// TIA Portal V15.1 export
// export: Created 2026-01-09T13:45:09.5933512Z, ExportSetting WithDefaults, WithReadOnly, DisplayName Totally Integrated Automation Portal, DisplayVersion V15.1 Update 8, DisplayName TIA Portal Openness, DisplayVersion V15.1 Update 8, DisplayName STEP 7 Professional, DisplayVersion V15.1 Update 8, DisplayName WinCC Advanced, DisplayVersion V15.1 Update 8
ORGANIZATION_BLOCK "Main_P1"   // OB1, LAD, ProgramCycle
TITLE = "Main Program Sweep (Cycle)"
{ S7_Optimized_Access := 'TRUE' }
VERSION : 0.1
// stored: AutoNumber true, CodeModifiedDate 2026-01-04T14:29:42.3003179Z, CompileDate 2026-01-04T14:29:49.7688293Z, ConstantName OB_Main_P1, CreationDate 2024-10-12T12:36:08.0193576Z, EventClass Program cycle, HandleErrorsWithinBlock false, InterfaceModifiedDate 2008-07-21T16:55:08.419547Z, IsConsistent true, IsIECCheckEnabled false, IsKnowHowProtected false, IsWriteProtected false, ModifiedDate 2026-01-04T14:29:42.3003179Z, ParameterModified 2008-07-21T16:55:08.419547Z, PLCSimAdvancedSupport false, PriorityNumber 1, ProcessImagePartNumber 65535, SetENOAutomatically False, StructureModified 2008-07-21T16:55:08.419547Z
   VAR_INPUT
      Initial_Call : Bool;   // Initial call of this OB
      Remanence : Bool;   // =True, if remanent data are available
   END_VAR
   VAR_TEMP   // added for the SCL form of the ladder/FBD networks
      _w1 : Bool;
      _w2 : Bool;
      _w3 : Bool;
      _w4 : Bool;
      _w5 : Bool;
      _w6 : Bool;
   END_VAR
BEGIN

REGION Network 1: MOVE INPUT
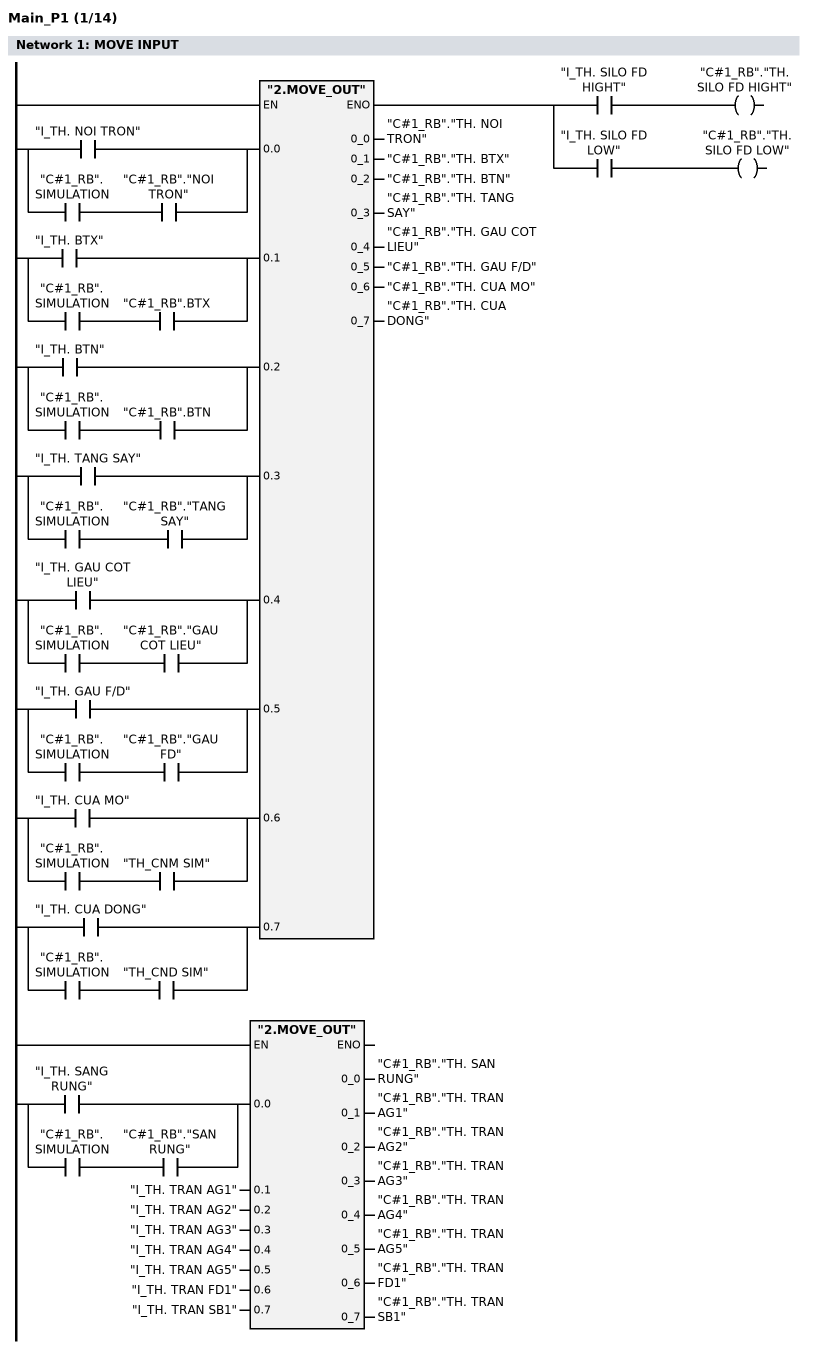
   RUNG wire#powerrail
      "2.MOVE_OUT"("0.0" := wire#w1, "0.1" := wire#w2, "0.2" := wire#w3, "0.3" := wire#w4, "0.4" := wire#w5, "0.5" := wire#w6, "0.6" := wire#w7, "0.7" := wire#w8, "0_0" => "C#1_RB"."TH. NOI TRON", "0_1" => "C#1_RB"."TH. BTX", "0_2" => "C#1_RB"."TH. BTN", "0_3" => "C#1_RB"."TH. TANG SAY", "0_4" => "C#1_RB"."TH. GAU COT LIEU", "0_5" => "C#1_RB"."TH. GAU F/D", "0_6" => "C#1_RB"."TH. CUA MO", "0_7" => "C#1_RB"."TH. CUA DONG")
      wire#w9
      Contact( "I_TH. SILO FD HIGHT" )
      Coil( "C#1_RB"."TH. SILO FD HIGHT" )
   END_RUNG
   RUNG wire#powerrail
      Contact( "I_TH. NOI TRON" )
   END_RUNG wire#w1
   RUNG wire#powerrail
      Contact( "C#1_RB".SIMULATION )
      Contact( "C#1_RB"."NOI TRON" )
   END_RUNG wire#w1
   RUNG wire#powerrail
      Contact( "I_TH. BTX" )
   END_RUNG wire#w2
   RUNG wire#powerrail
      Contact( "C#1_RB".SIMULATION )
      Contact( "C#1_RB".BTX )
   END_RUNG wire#w2
   RUNG wire#powerrail
      Contact( "I_TH. BTN" )
   END_RUNG wire#w3
   RUNG wire#powerrail
      Contact( "C#1_RB".SIMULATION )
      Contact( "C#1_RB".BTN )
   END_RUNG wire#w3
   RUNG wire#powerrail
      Contact( "I_TH. TANG SAY" )
   END_RUNG wire#w4
   RUNG wire#powerrail
      Contact( "C#1_RB".SIMULATION )
      Contact( "C#1_RB"."TANG SAY" )
   END_RUNG wire#w4
   RUNG wire#powerrail
      Contact( "I_TH. GAU COT LIEU" )
   END_RUNG wire#w5
   RUNG wire#powerrail
      Contact( "C#1_RB".SIMULATION )
      Contact( "C#1_RB"."GAU COT LIEU" )
   END_RUNG wire#w5
   RUNG wire#powerrail
      Contact( "I_TH. GAU F/D" )
   END_RUNG wire#w6
   RUNG wire#powerrail
      Contact( "C#1_RB".SIMULATION )
      Contact( "C#1_RB"."GAU FD" )
   END_RUNG wire#w6
   RUNG wire#powerrail
      Contact( "I_TH. CUA MO" )
   END_RUNG wire#w7
   RUNG wire#powerrail
      Contact( "C#1_RB".SIMULATION )
      Contact( "TH_CNM SIM" )
   END_RUNG wire#w7
   RUNG wire#powerrail
      Contact( "I_TH. CUA DONG" )
   END_RUNG wire#w8
   RUNG wire#powerrail
      Contact( "C#1_RB".SIMULATION )
      Contact( "TH_CND SIM" )
   END_RUNG wire#w8
   RUNG wire#w9
      Contact( "I_TH. SILO FD LOW" )
      Coil( "C#1_RB"."TH. SILO FD LOW" )
   END_RUNG
   RUNG wire#powerrail
      "2.MOVE_OUT"("0.0" := wire#w10, "0.1" := "I_TH. TRAN AG1", "0.2" := "I_TH. TRAN AG2", "0.3" := "I_TH. TRAN AG3", "0.4" := "I_TH. TRAN AG4", "0.5" := "I_TH. TRAN AG5", "0.6" := "I_TH. TRAN FD1", "0.7" := "I_TH. TRAN SB1", "0_0" => "C#1_RB"."TH. SAN RUNG", "0_1" => "C#1_RB"."TH. TRAN AG1", "0_2" => "C#1_RB"."TH. TRAN AG2", "0_3" => "C#1_RB"."TH. TRAN AG3", "0_4" => "C#1_RB"."TH. TRAN AG4", "0_5" => "C#1_RB"."TH. TRAN AG5", "0_6" => "C#1_RB"."TH. TRAN FD1", "0_7" => "C#1_RB"."TH. TRAN SB1")
   END_RUNG
   RUNG wire#powerrail
      Contact( "I_TH. SANG RUNG" )
   END_RUNG wire#w10
   RUNG wire#powerrail
      Contact( "C#1_RB".SIMULATION )
      Contact( "C#1_RB"."SAN RUNG" )
   END_RUNG wire#w10
   // the same network as SCL:
   "2.MOVE_OUT"("0.0" := "I_TH. NOI TRON" OR ("C#1_RB".SIMULATION AND "C#1_RB"."NOI TRON"),
                "0.1" := "I_TH. BTX" OR ("C#1_RB".SIMULATION AND "C#1_RB".BTX),
                "0.2" := "I_TH. BTN" OR ("C#1_RB".SIMULATION AND "C#1_RB".BTN),
                "0.3" := "I_TH. TANG SAY" OR ("C#1_RB".SIMULATION AND "C#1_RB"."TANG SAY"),
                "0.4" := "I_TH. GAU COT LIEU" OR ("C#1_RB".SIMULATION AND "C#1_RB"."GAU COT LIEU"),
                "0.5" := "I_TH. GAU F/D" OR ("C#1_RB".SIMULATION AND "C#1_RB"."GAU FD"),
                "0.6" := "I_TH. CUA MO" OR ("C#1_RB".SIMULATION AND "TH_CNM SIM"),
                "0.7" := "I_TH. CUA DONG" OR ("C#1_RB".SIMULATION AND "TH_CND SIM"),
                "0_0" => "C#1_RB"."TH. NOI TRON",
                "0_1" => "C#1_RB"."TH. BTX",
                "0_2" => "C#1_RB"."TH. BTN",
                "0_3" => "C#1_RB"."TH. TANG SAY",
                "0_4" => "C#1_RB"."TH. GAU COT LIEU",
                "0_5" => "C#1_RB"."TH. GAU F/D",
                "0_6" => "C#1_RB"."TH. CUA MO",
                "0_7" => "C#1_RB"."TH. CUA DONG",
                ENO => #_w1);
   "C#1_RB"."TH. SILO FD HIGHT" := #_w1 AND "I_TH. SILO FD HIGHT";
   "C#1_RB"."TH. SILO FD LOW" := #_w1 AND "I_TH. SILO FD LOW";
   "2.MOVE_OUT"("0.0" := "I_TH. SANG RUNG" OR ("C#1_RB".SIMULATION AND "C#1_RB"."SAN RUNG"),
                "0.1" := "I_TH. TRAN AG1",
                "0.2" := "I_TH. TRAN AG2",
                "0.3" := "I_TH. TRAN AG3",
                "0.4" := "I_TH. TRAN AG4",
                "0.5" := "I_TH. TRAN AG5",
                "0.6" := "I_TH. TRAN FD1",
                "0.7" := "I_TH. TRAN SB1",
                "0_0" => "C#1_RB"."TH. SAN RUNG",
                "0_1" => "C#1_RB"."TH. TRAN AG1",
                "0_2" => "C#1_RB"."TH. TRAN AG2",
                "0_3" => "C#1_RB"."TH. TRAN AG3",
                "0_4" => "C#1_RB"."TH. TRAN AG4",
                "0_5" => "C#1_RB"."TH. TRAN AG5",
                "0_6" => "C#1_RB"."TH. TRAN FD1",
                "0_7" => "C#1_RB"."TH. TRAN SB1");
END_REGION

REGION Network 2: MOVE OUTPUT
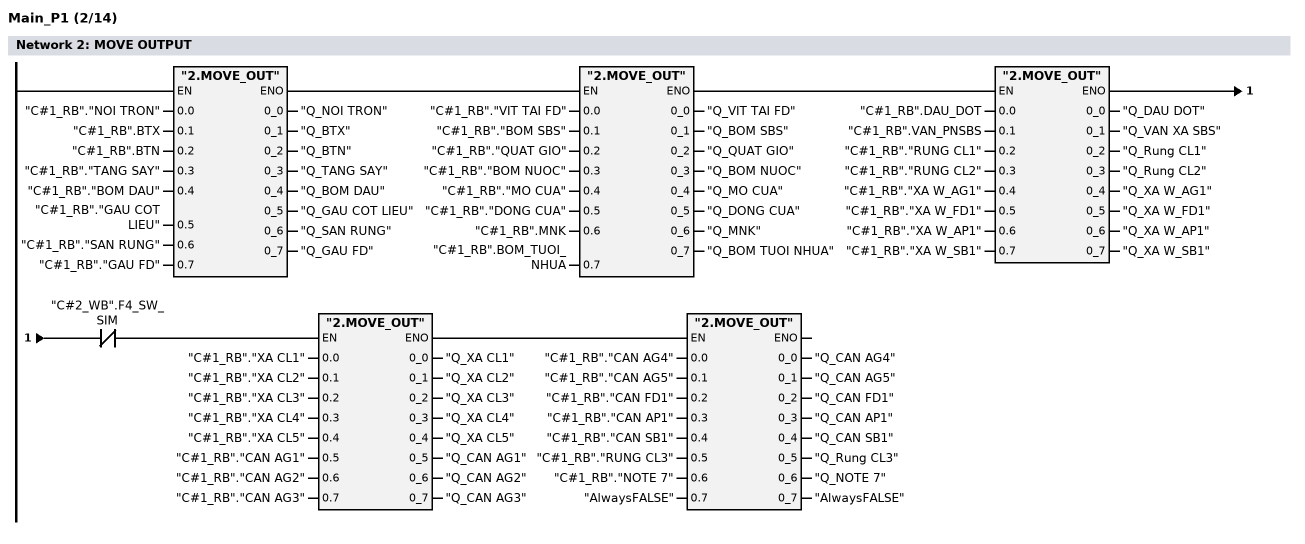
   RUNG wire#powerrail
      "2.MOVE_OUT"("0.0" := "C#1_RB"."NOI TRON", "0.1" := "C#1_RB".BTX, "0.2" := "C#1_RB".BTN, "0.3" := "C#1_RB"."TANG SAY", "0.4" := "C#1_RB"."BOM DAU", "0.5" := "C#1_RB"."GAU COT LIEU", "0.6" := "C#1_RB"."SAN RUNG", "0.7" := "C#1_RB"."GAU FD", "0_0" => "Q_NOI TRON", "0_1" => "Q_BTX", "0_2" => "Q_BTN", "0_3" => "Q_TANG SAY", "0_4" => "Q_BOM DAU", "0_5" => "Q_GAU COT LIEU", "0_6" => "Q_SAN RUNG", "0_7" => "Q_GAU FD")
      "2.MOVE_OUT"("0.0" := "C#1_RB"."VIT TAI FD", "0.1" := "C#1_RB"."BOM SBS", "0.2" := "C#1_RB"."QUAT GIO", "0.3" := "C#1_RB"."BOM NUOC", "0.4" := "C#1_RB"."MO CUA", "0.5" := "C#1_RB"."DONG CUA", "0.6" := "C#1_RB".MNK, "0.7" := "C#1_RB".BOM_TUOI_NHUA, "0_0" => "Q_VIT TAI FD", "0_1" => "Q_BOM SBS", "0_2" => "Q_QUAT GIO", "0_3" => "Q_BOM NUOC", "0_4" => "Q_MO CUA", "0_5" => "Q_DONG CUA", "0_6" => "Q_MNK", "0_7" => "Q_BOM TUOI NHUA")
      "2.MOVE_OUT"("0.0" := "C#1_RB".DAU_DOT, "0.1" := "C#1_RB".VAN_PNSBS, "0.2" := "C#1_RB"."RUNG CL1", "0.3" := "C#1_RB"."RUNG CL2", "0.4" := "C#1_RB"."XA W_AG1", "0.5" := "C#1_RB"."XA W_FD1", "0.6" := "C#1_RB"."XA W_AP1", "0.7" := "C#1_RB"."XA W_SB1", "0_0" => "Q_DAU DOT", "0_1" => "Q_VAN XA SBS", "0_2" => "Q_Rung CL1", "0_3" => "Q_Rung CL2", "0_4" => "Q_XA W_AG1", "0_5" => "Q_XA W_FD1", "0_6" => "Q_XA W_AP1", "0_7" => "Q_XA W_SB1")
      I_Contact( "C#2_WB".F4_SW_SIM )
      "2.MOVE_OUT"("0.0" := "C#1_RB"."XA CL1", "0.1" := "C#1_RB"."XA CL2", "0.2" := "C#1_RB"."XA CL3", "0.3" := "C#1_RB"."XA CL4", "0.4" := "C#1_RB"."XA CL5", "0.5" := "C#1_RB"."CAN AG1", "0.6" := "C#1_RB"."CAN AG2", "0.7" := "C#1_RB"."CAN AG3", "0_0" => "Q_XA CL1", "0_1" => "Q_XA CL2", "0_2" => "Q_XA CL3", "0_3" => "Q_XA CL4", "0_4" => "Q_XA CL5", "0_5" => "Q_CAN AG1", "0_6" => "Q_CAN AG2", "0_7" => "Q_CAN AG3")
      "2.MOVE_OUT"("0.0" := "C#1_RB"."CAN AG4", "0.1" := "C#1_RB"."CAN AG5", "0.2" := "C#1_RB"."CAN FD1", "0.3" := "C#1_RB"."CAN AP1", "0.4" := "C#1_RB"."CAN SB1", "0.5" := "C#1_RB"."RUNG CL3", "0.6" := "C#1_RB"."NOTE 7", "0.7" := "AlwaysFALSE", "0_0" => "Q_CAN AG4", "0_1" => "Q_CAN AG5", "0_2" => "Q_CAN FD1", "0_3" => "Q_CAN AP1", "0_4" => "Q_CAN SB1", "0_5" => "Q_Rung CL3", "0_6" => "Q_NOTE 7", "0_7" => "AlwaysFALSE")
   END_RUNG
   // the same network as SCL:
   "2.MOVE_OUT"("0.0" := "C#1_RB"."NOI TRON",
                "0.1" := "C#1_RB".BTX,
                "0.2" := "C#1_RB".BTN,
                "0.3" := "C#1_RB"."TANG SAY",
                "0.4" := "C#1_RB"."BOM DAU",
                "0.5" := "C#1_RB"."GAU COT LIEU",
                "0.6" := "C#1_RB"."SAN RUNG",
                "0.7" := "C#1_RB"."GAU FD",
                "0_0" => "Q_NOI TRON",
                "0_1" => "Q_BTX",
                "0_2" => "Q_BTN",
                "0_3" => "Q_TANG SAY",
                "0_4" => "Q_BOM DAU",
                "0_5" => "Q_GAU COT LIEU",
                "0_6" => "Q_SAN RUNG",
                "0_7" => "Q_GAU FD",
                ENO => #_w1);
   "2.MOVE_OUT"(EN := #_w1,
                "0.0" := "C#1_RB"."VIT TAI FD",
                "0.1" := "C#1_RB"."BOM SBS",
                "0.2" := "C#1_RB"."QUAT GIO",
                "0.3" := "C#1_RB"."BOM NUOC",
                "0.4" := "C#1_RB"."MO CUA",
                "0.5" := "C#1_RB"."DONG CUA",
                "0.6" := "C#1_RB".MNK,
                "0.7" := "C#1_RB".BOM_TUOI_NHUA,
                "0_0" => "Q_VIT TAI FD",
                "0_1" => "Q_BOM SBS",
                "0_2" => "Q_QUAT GIO",
                "0_3" => "Q_BOM NUOC",
                "0_4" => "Q_MO CUA",
                "0_5" => "Q_DONG CUA",
                "0_6" => "Q_MNK",
                "0_7" => "Q_BOM TUOI NHUA",
                ENO => #_w2);
   "2.MOVE_OUT"(EN := #_w2,
                "0.0" := "C#1_RB".DAU_DOT,
                "0.1" := "C#1_RB".VAN_PNSBS,
                "0.2" := "C#1_RB"."RUNG CL1",
                "0.3" := "C#1_RB"."RUNG CL2",
                "0.4" := "C#1_RB"."XA W_AG1",
                "0.5" := "C#1_RB"."XA W_FD1",
                "0.6" := "C#1_RB"."XA W_AP1",
                "0.7" := "C#1_RB"."XA W_SB1",
                "0_0" => "Q_DAU DOT",
                "0_1" => "Q_VAN XA SBS",
                "0_2" => "Q_Rung CL1",
                "0_3" => "Q_Rung CL2",
                "0_4" => "Q_XA W_AG1",
                "0_5" => "Q_XA W_FD1",
                "0_6" => "Q_XA W_AP1",
                "0_7" => "Q_XA W_SB1",
                ENO => #_w3);
   "2.MOVE_OUT"(EN := #_w3 AND NOT "C#2_WB".F4_SW_SIM,
                "0.0" := "C#1_RB"."XA CL1",
                "0.1" := "C#1_RB"."XA CL2",
                "0.2" := "C#1_RB"."XA CL3",
                "0.3" := "C#1_RB"."XA CL4",
                "0.4" := "C#1_RB"."XA CL5",
                "0.5" := "C#1_RB"."CAN AG1",
                "0.6" := "C#1_RB"."CAN AG2",
                "0.7" := "C#1_RB"."CAN AG3",
                "0_0" => "Q_XA CL1",
                "0_1" => "Q_XA CL2",
                "0_2" => "Q_XA CL3",
                "0_3" => "Q_XA CL4",
                "0_4" => "Q_XA CL5",
                "0_5" => "Q_CAN AG1",
                "0_6" => "Q_CAN AG2",
                "0_7" => "Q_CAN AG3",
                ENO => #_w4);
   IF #_w4 THEN
       "2.MOVE_OUT"("0.0" := "C#1_RB"."CAN AG4",
                    "0.1" := "C#1_RB"."CAN AG5",
                    "0.2" := "C#1_RB"."CAN FD1",
                    "0.3" := "C#1_RB"."CAN AP1",
                    "0.4" := "C#1_RB"."CAN SB1",
                    "0.5" := "C#1_RB"."RUNG CL3",
                    "0.6" := "C#1_RB"."NOTE 7",
                    "0.7" := "AlwaysFALSE",
                    "0_0" => "Q_CAN AG4",
                    "0_1" => "Q_CAN AG5",
                    "0_2" => "Q_CAN FD1",
                    "0_3" => "Q_CAN AP1",
                    "0_4" => "Q_CAN SB1",
                    "0_5" => "Q_Rung CL3",
                    "0_6" => "Q_NOTE 7",
                    "0_7" => "AlwaysFALSE");
   END_IF;
END_REGION

REGION Network 3: ĐIỀU KHIỂN TAY
   // Nếu ở chế độ Tự động, mà TANG SẤY chưa được mở thì không bật được Băng tải xiêng, tương tự nếu chưa mở BTX thì không mở được BTN
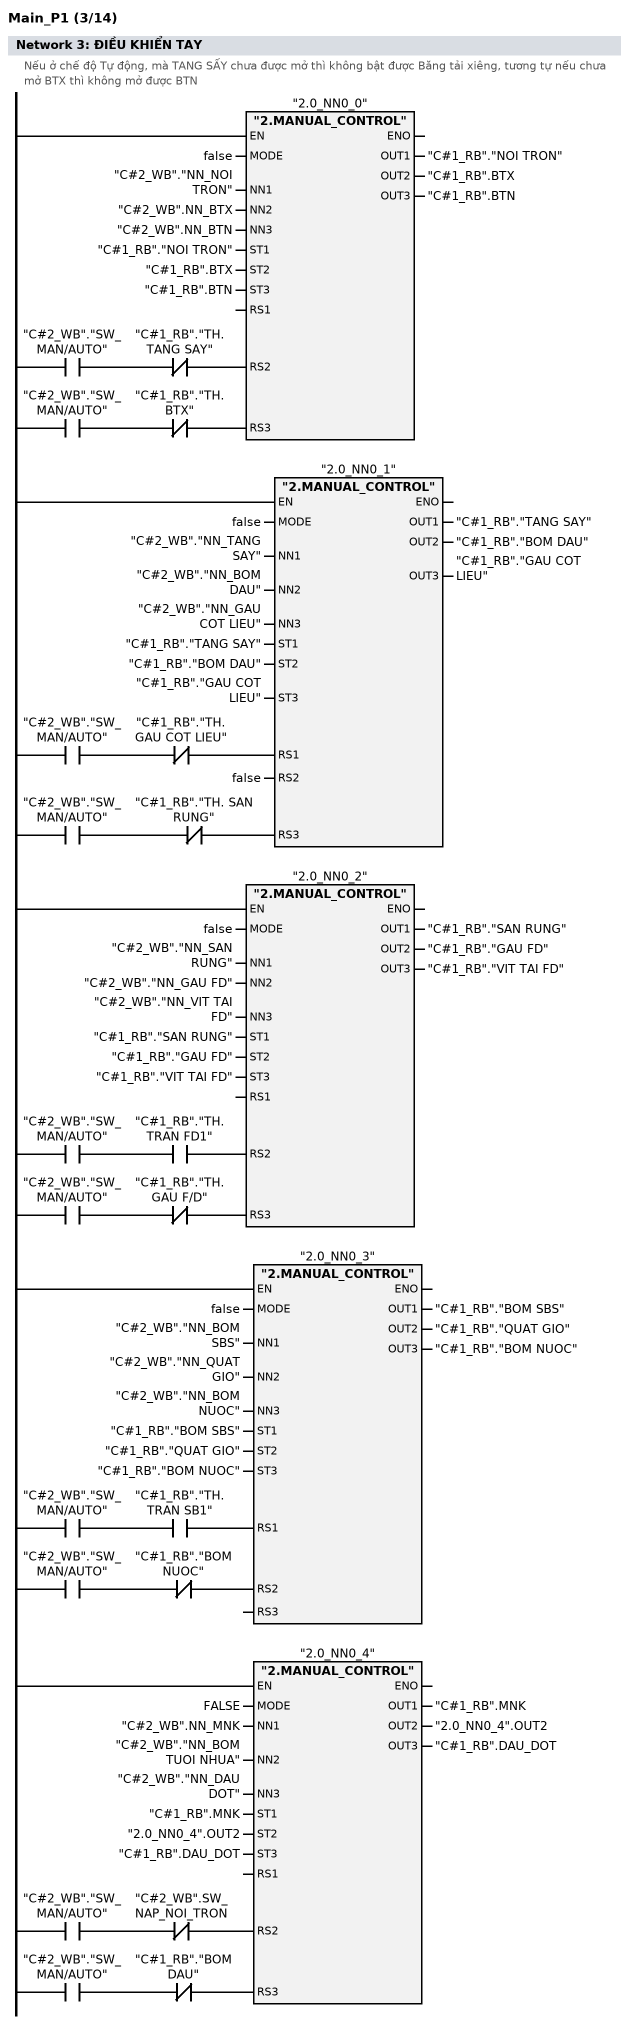
   RUNG wire#powerrail
      "2.0_NN0_0"(RS2 := wire#w1, RS3 := wire#w2, MODE := false, NN1 := "C#2_WB"."NN_NOI TRON", NN2 := "C#2_WB".NN_BTX, NN3 := "C#2_WB".NN_BTN, ST1 := "C#1_RB"."NOI TRON", ST2 := "C#1_RB".BTX, ST3 := "C#1_RB".BTN, RS1 :=, OUT1 => "C#1_RB"."NOI TRON", OUT2 => "C#1_RB".BTX, OUT3 => "C#1_RB".BTN)
   END_RUNG
   RUNG wire#powerrail
      Contact( "C#2_WB"."SW_MAN/AUTO" )
      I_Contact( "C#1_RB"."TH. TANG SAY" )
   END_RUNG wire#w1
   RUNG wire#powerrail
      Contact( "C#2_WB"."SW_MAN/AUTO" )
      I_Contact( "C#1_RB"."TH. BTX" )
   END_RUNG wire#w2
   RUNG wire#powerrail
      "2.0_NN0_1"(RS1 := wire#w3, RS3 := wire#w4, MODE := false, NN1 := "C#2_WB"."NN_TANG SAY", NN2 := "C#2_WB"."NN_BOM DAU", NN3 := "C#2_WB"."NN_GAU COT LIEU", ST1 := "C#1_RB"."TANG SAY", ST2 := "C#1_RB"."BOM DAU", ST3 := "C#1_RB"."GAU COT LIEU", RS2 := false, OUT1 => "C#1_RB"."TANG SAY", OUT2 => "C#1_RB"."BOM DAU", OUT3 => "C#1_RB"."GAU COT LIEU")
   END_RUNG
   RUNG wire#powerrail
      Contact( "C#2_WB"."SW_MAN/AUTO" )
      I_Contact( "C#1_RB"."TH. GAU COT LIEU" )
   END_RUNG wire#w3
   RUNG wire#powerrail
      Contact( "C#2_WB"."SW_MAN/AUTO" )
      I_Contact( "C#1_RB"."TH. SAN RUNG" )
   END_RUNG wire#w4
   RUNG wire#powerrail
      "2.0_NN0_2"(RS2 := wire#w5, RS3 := wire#w6, MODE := false, NN1 := "C#2_WB"."NN_SAN RUNG", NN2 := "C#2_WB"."NN_GAU FD", NN3 := "C#2_WB"."NN_VIT TAI FD", ST1 := "C#1_RB"."SAN RUNG", ST2 := "C#1_RB"."GAU FD", ST3 := "C#1_RB"."VIT TAI FD", RS1 :=, OUT1 => "C#1_RB"."SAN RUNG", OUT2 => "C#1_RB"."GAU FD", OUT3 => "C#1_RB"."VIT TAI FD")
   END_RUNG
   RUNG wire#powerrail
      Contact( "C#2_WB"."SW_MAN/AUTO" )
      Contact( "C#1_RB"."TH. TRAN FD1" )
   END_RUNG wire#w5
   RUNG wire#powerrail
      Contact( "C#2_WB"."SW_MAN/AUTO" )
      I_Contact( "C#1_RB"."TH. GAU F/D" )
   END_RUNG wire#w6
   RUNG wire#powerrail
      "2.0_NN0_3"(RS1 := wire#w7, RS2 := wire#w8, MODE := false, NN1 := "C#2_WB"."NN_BOM SBS", NN2 := "C#2_WB"."NN_QUAT GIO", NN3 := "C#2_WB"."NN_BOM NUOC", ST1 := "C#1_RB"."BOM SBS", ST2 := "C#1_RB"."QUAT GIO", ST3 := "C#1_RB"."BOM NUOC", RS3 :=, OUT1 => "C#1_RB"."BOM SBS", OUT2 => "C#1_RB"."QUAT GIO", OUT3 => "C#1_RB"."BOM NUOC")
   END_RUNG
   RUNG wire#powerrail
      Contact( "C#2_WB"."SW_MAN/AUTO" )
      Contact( "C#1_RB"."TH. TRAN SB1" )
   END_RUNG wire#w7
   RUNG wire#powerrail
      Contact( "C#2_WB"."SW_MAN/AUTO" )
      I_Contact( "C#1_RB"."BOM NUOC" )
   END_RUNG wire#w8
   RUNG wire#powerrail
      "2.0_NN0_4"(RS2 := wire#w9, RS3 := wire#w10, MODE := FALSE, NN1 := "C#2_WB".NN_MNK, NN2 := "C#2_WB"."NN_BOM TUOI NHUA", NN3 := "C#2_WB"."NN_DAU DOT", ST1 := "C#1_RB".MNK, ST2 := "2.0_NN0_4".OUT2, ST3 := "C#1_RB".DAU_DOT, RS1 :=, OUT1 => "C#1_RB".MNK, OUT2 => "2.0_NN0_4".OUT2, OUT3 => "C#1_RB".DAU_DOT)
   END_RUNG
   RUNG wire#powerrail
      Contact( "C#2_WB"."SW_MAN/AUTO" )
      I_Contact( "C#2_WB".SW_NAP_NOI_TRON )
   END_RUNG wire#w9
   RUNG wire#powerrail
      Contact( "C#2_WB"."SW_MAN/AUTO" )
      I_Contact( "C#1_RB"."BOM DAU" )
   END_RUNG wire#w10
   // the same network as SCL:
   "2.0_NN0_0"(MODE := false,   // "2.MANUAL_CONTROL"
               NN1 := "C#2_WB"."NN_NOI TRON",
               NN2 := "C#2_WB".NN_BTX,
               NN3 := "C#2_WB".NN_BTN,
               ST1 := "C#1_RB"."NOI TRON",
               ST2 := "C#1_RB".BTX,
               ST3 := "C#1_RB".BTN,
               RS2 := "C#2_WB"."SW_MAN/AUTO" AND NOT "C#1_RB"."TH. TANG SAY",
               RS3 := "C#2_WB"."SW_MAN/AUTO" AND NOT "C#1_RB"."TH. BTX",
               OUT1 => "C#1_RB"."NOI TRON",
               OUT2 => "C#1_RB".BTX,
               OUT3 => "C#1_RB".BTN);
   "2.0_NN0_1"(MODE := false,   // "2.MANUAL_CONTROL"
               NN1 := "C#2_WB"."NN_TANG SAY",
               NN2 := "C#2_WB"."NN_BOM DAU",
               NN3 := "C#2_WB"."NN_GAU COT LIEU",
               ST1 := "C#1_RB"."TANG SAY",
               ST2 := "C#1_RB"."BOM DAU",
               ST3 := "C#1_RB"."GAU COT LIEU",
               RS1 := "C#2_WB"."SW_MAN/AUTO" AND NOT "C#1_RB"."TH. GAU COT LIEU",
               RS2 := false,
               RS3 := "C#2_WB"."SW_MAN/AUTO" AND NOT "C#1_RB"."TH. SAN RUNG",
               OUT1 => "C#1_RB"."TANG SAY",
               OUT2 => "C#1_RB"."BOM DAU",
               OUT3 => "C#1_RB"."GAU COT LIEU");
   "2.0_NN0_2"(MODE := false,   // "2.MANUAL_CONTROL"
               NN1 := "C#2_WB"."NN_SAN RUNG",
               NN2 := "C#2_WB"."NN_GAU FD",
               NN3 := "C#2_WB"."NN_VIT TAI FD",
               ST1 := "C#1_RB"."SAN RUNG",
               ST2 := "C#1_RB"."GAU FD",
               ST3 := "C#1_RB"."VIT TAI FD",
               RS2 := "C#2_WB"."SW_MAN/AUTO" AND "C#1_RB"."TH. TRAN FD1",
               RS3 := "C#2_WB"."SW_MAN/AUTO" AND NOT "C#1_RB"."TH. GAU F/D",
               OUT1 => "C#1_RB"."SAN RUNG",
               OUT2 => "C#1_RB"."GAU FD",
               OUT3 => "C#1_RB"."VIT TAI FD");
   "2.0_NN0_3"(MODE := false,   // "2.MANUAL_CONTROL"
               NN1 := "C#2_WB"."NN_BOM SBS",
               NN2 := "C#2_WB"."NN_QUAT GIO",
               NN3 := "C#2_WB"."NN_BOM NUOC",
               ST1 := "C#1_RB"."BOM SBS",
               ST2 := "C#1_RB"."QUAT GIO",
               ST3 := "C#1_RB"."BOM NUOC",
               RS1 := "C#2_WB"."SW_MAN/AUTO" AND "C#1_RB"."TH. TRAN SB1",
               RS2 := "C#2_WB"."SW_MAN/AUTO" AND NOT "C#1_RB"."BOM NUOC",
               OUT1 => "C#1_RB"."BOM SBS",
               OUT2 => "C#1_RB"."QUAT GIO",
               OUT3 => "C#1_RB"."BOM NUOC");
   "2.0_NN0_4"(MODE := FALSE,   // "2.MANUAL_CONTROL"
               NN1 := "C#2_WB".NN_MNK,
               NN2 := "C#2_WB"."NN_BOM TUOI NHUA",
               NN3 := "C#2_WB"."NN_DAU DOT",
               ST1 := "C#1_RB".MNK,
               ST2 := "2.0_NN0_4".OUT2,
               ST3 := "C#1_RB".DAU_DOT,
               RS2 := "C#2_WB"."SW_MAN/AUTO" AND NOT "C#2_WB".SW_NAP_NOI_TRON,
               RS3 := "C#2_WB"."SW_MAN/AUTO" AND NOT "C#1_RB"."BOM DAU",
               OUT1 => "C#1_RB".MNK,
               OUT2 => "2.0_NN0_4".OUT2,
               OUT3 => "C#1_RB".DAU_DOT);
END_REGION

REGION Network 4: CONVERT ANALOG IN PUT (0.0/ 0-10V: 1.0/4-20mA: 2.0/0-20mA)
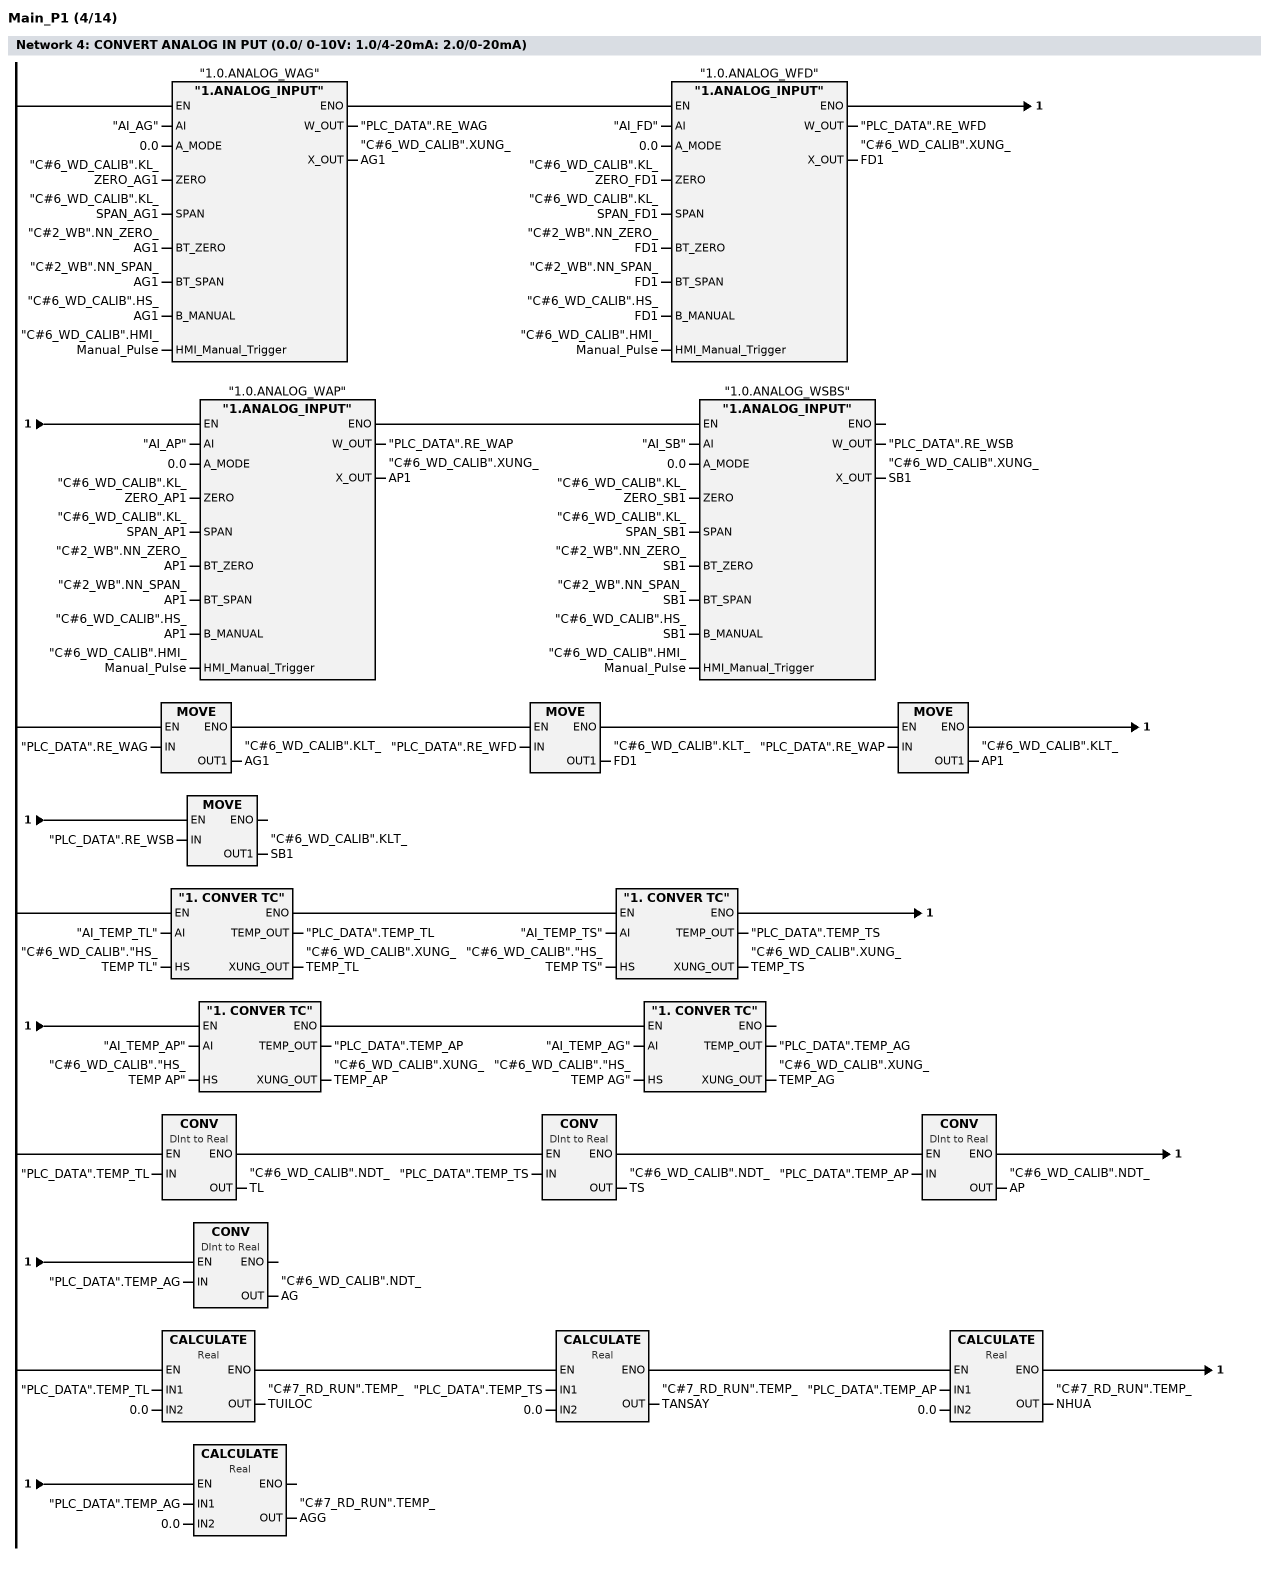
   RUNG wire#powerrail
      "1.0.ANALOG_WAG"(AI := "AI_AG", A_MODE := 0.0, ZERO := "C#6_WD_CALIB".KL_ZERO_AG1, SPAN := "C#6_WD_CALIB".KL_SPAN_AG1, BT_ZERO := "C#2_WB".NN_ZERO_AG1, BT_SPAN := "C#2_WB".NN_SPAN_AG1, B_MANUAL := "C#6_WD_CALIB".HS_AG1, HMI_Manual_Trigger := "C#6_WD_CALIB".HMI_Manual_Pulse, W_OUT => "PLC_DATA".RE_WAG, X_OUT => "C#6_WD_CALIB".XUNG_AG1)
      "1.0.ANALOG_WFD"(AI := "AI_FD", A_MODE := 0.0, ZERO := "C#6_WD_CALIB".KL_ZERO_FD1, SPAN := "C#6_WD_CALIB".KL_SPAN_FD1, BT_ZERO := "C#2_WB".NN_ZERO_FD1, BT_SPAN := "C#2_WB".NN_SPAN_FD1, B_MANUAL := "C#6_WD_CALIB".HS_FD1, HMI_Manual_Trigger := "C#6_WD_CALIB".HMI_Manual_Pulse, W_OUT => "PLC_DATA".RE_WFD, X_OUT => "C#6_WD_CALIB".XUNG_FD1)
      "1.0.ANALOG_WAP"(AI := "AI_AP", A_MODE := 0.0, ZERO := "C#6_WD_CALIB".KL_ZERO_AP1, SPAN := "C#6_WD_CALIB".KL_SPAN_AP1, BT_ZERO := "C#2_WB".NN_ZERO_AP1, BT_SPAN := "C#2_WB".NN_SPAN_AP1, B_MANUAL := "C#6_WD_CALIB".HS_AP1, HMI_Manual_Trigger := "C#6_WD_CALIB".HMI_Manual_Pulse, W_OUT => "PLC_DATA".RE_WAP, X_OUT => "C#6_WD_CALIB".XUNG_AP1)
      "1.0.ANALOG_WSBS"(AI := "AI_SB", A_MODE := 0.0, ZERO := "C#6_WD_CALIB".KL_ZERO_SB1, SPAN := "C#6_WD_CALIB".KL_SPAN_SB1, BT_ZERO := "C#2_WB".NN_ZERO_SB1, BT_SPAN := "C#2_WB".NN_SPAN_SB1, B_MANUAL := "C#6_WD_CALIB".HS_SB1, HMI_Manual_Trigger := "C#6_WD_CALIB".HMI_Manual_Pulse, W_OUT => "PLC_DATA".RE_WSB, X_OUT => "C#6_WD_CALIB".XUNG_SB1)
   END_RUNG
   RUNG wire#powerrail
      { S7_GenerateENO := "TRUE" } Move(in := "PLC_DATA".RE_WAG, out1 => "C#6_WD_CALIB".KLT_AG1)
      { S7_GenerateENO := "TRUE" } Move(in := "PLC_DATA".RE_WFD, out1 => "C#6_WD_CALIB".KLT_FD1)
      { S7_GenerateENO := "TRUE" } Move(in := "PLC_DATA".RE_WAP, out1 => "C#6_WD_CALIB".KLT_AP1)
      { S7_GenerateENO := "TRUE" } Move(in := "PLC_DATA".RE_WSB, out1 => "C#6_WD_CALIB".KLT_SB1)
   END_RUNG
   RUNG wire#powerrail
      "1. CONVER TC"(AI := "AI_TEMP_TL", HS := "C#6_WD_CALIB"."HS_TEMP TL", TEMP_OUT => "PLC_DATA".TEMP_TL, XUNG_OUT => "C#6_WD_CALIB".XUNG_TEMP_TL)
      "1. CONVER TC"(AI := "AI_TEMP_TS", HS := "C#6_WD_CALIB"."HS_TEMP TS", TEMP_OUT => "PLC_DATA".TEMP_TS, XUNG_OUT => "C#6_WD_CALIB".XUNG_TEMP_TS)
      "1. CONVER TC"(AI := "AI_TEMP_AP", HS := "C#6_WD_CALIB"."HS_TEMP AP", TEMP_OUT => "PLC_DATA".TEMP_AP, XUNG_OUT => "C#6_WD_CALIB".XUNG_TEMP_AP)
      "1. CONVER TC"(AI := "AI_TEMP_AG", HS := "C#6_WD_CALIB"."HS_TEMP AG", TEMP_OUT => "PLC_DATA".TEMP_AG, XUNG_OUT => "C#6_WD_CALIB".XUNG_TEMP_AG)
   END_RUNG
   RUNG wire#powerrail
      { S7_Templates := "[SrcType := DInt, DestType := Real]" } Convert(in := "PLC_DATA".TEMP_TL, out => "C#6_WD_CALIB".NDT_TL)
      { S7_Templates := "[SrcType := DInt, DestType := Real]" } Convert(in := "PLC_DATA".TEMP_TS, out => "C#6_WD_CALIB".NDT_TS)
      { S7_Templates := "[SrcType := DInt, DestType := Real]" } Convert(in := "PLC_DATA".TEMP_AP, out => "C#6_WD_CALIB".NDT_AP)
      { S7_Templates := "[SrcType := DInt, DestType := Real]" } Convert(in := "PLC_DATA".TEMP_AG, out => "C#6_WD_CALIB".NDT_AG)
   END_RUNG
   RUNG wire#powerrail
      { S7_Templates := "SrcType := Real"; S7_Expression := "IN1+IN2" } Calculate(in1 := "PLC_DATA".TEMP_TL, in2 := 0.0, out => "C#7_RD_RUN".TEMP_TUILOC)
      { S7_Templates := "SrcType := Real"; S7_Expression := "IN1+IN2" } Calculate(in1 := "PLC_DATA".TEMP_TS, in2 := 0.0, out => "C#7_RD_RUN".TEMP_TANSAY)
      { S7_Templates := "SrcType := Real"; S7_Expression := "IN1+IN2" } Calculate(in1 := "PLC_DATA".TEMP_AP, in2 := 0.0, out => "C#7_RD_RUN".TEMP_NHUA)
      { S7_Templates := "SrcType := Real"; S7_Expression := "IN1+IN2" } Calculate(in1 := "PLC_DATA".TEMP_AG, in2 := 0.0, out => "C#7_RD_RUN".TEMP_AGG)
   END_RUNG
   // the same network as SCL:
   // ENO of a box is taken as its EN; it also drops when the box reports an error
   "1.0.ANALOG_WAG"(AI := "AI_AG",   // "1.ANALOG_INPUT"
                    A_MODE := 0.0,
                    ZERO := "C#6_WD_CALIB".KL_ZERO_AG1,
                    SPAN := "C#6_WD_CALIB".KL_SPAN_AG1,
                    BT_ZERO := "C#2_WB".NN_ZERO_AG1,
                    BT_SPAN := "C#2_WB".NN_SPAN_AG1,
                    B_MANUAL := "C#6_WD_CALIB".HS_AG1,
                    HMI_Manual_Trigger := "C#6_WD_CALIB".HMI_Manual_Pulse,
                    W_OUT => "PLC_DATA".RE_WAG,
                    X_OUT => "C#6_WD_CALIB".XUNG_AG1,
                    ENO => #_w1);
   "1.0.ANALOG_WFD"(EN := #_w1,   // "1.ANALOG_INPUT"
                    AI := "AI_FD",
                    A_MODE := 0.0,
                    ZERO := "C#6_WD_CALIB".KL_ZERO_FD1,
                    SPAN := "C#6_WD_CALIB".KL_SPAN_FD1,
                    BT_ZERO := "C#2_WB".NN_ZERO_FD1,
                    BT_SPAN := "C#2_WB".NN_SPAN_FD1,
                    B_MANUAL := "C#6_WD_CALIB".HS_FD1,
                    HMI_Manual_Trigger := "C#6_WD_CALIB".HMI_Manual_Pulse,
                    W_OUT => "PLC_DATA".RE_WFD,
                    X_OUT => "C#6_WD_CALIB".XUNG_FD1,
                    ENO => #_w2);
   "1.0.ANALOG_WAP"(EN := #_w2,   // "1.ANALOG_INPUT"
                    AI := "AI_AP",
                    A_MODE := 0.0,
                    ZERO := "C#6_WD_CALIB".KL_ZERO_AP1,
                    SPAN := "C#6_WD_CALIB".KL_SPAN_AP1,
                    BT_ZERO := "C#2_WB".NN_ZERO_AP1,
                    BT_SPAN := "C#2_WB".NN_SPAN_AP1,
                    B_MANUAL := "C#6_WD_CALIB".HS_AP1,
                    HMI_Manual_Trigger := "C#6_WD_CALIB".HMI_Manual_Pulse,
                    W_OUT => "PLC_DATA".RE_WAP,
                    X_OUT => "C#6_WD_CALIB".XUNG_AP1,
                    ENO => #_w3);
   IF #_w3 THEN
       "1.0.ANALOG_WSBS"(AI := "AI_SB",   // "1.ANALOG_INPUT"
                         A_MODE := 0.0,
                         ZERO := "C#6_WD_CALIB".KL_ZERO_SB1,
                         SPAN := "C#6_WD_CALIB".KL_SPAN_SB1,
                         BT_ZERO := "C#2_WB".NN_ZERO_SB1,
                         BT_SPAN := "C#2_WB".NN_SPAN_SB1,
                         B_MANUAL := "C#6_WD_CALIB".HS_SB1,
                         HMI_Manual_Trigger := "C#6_WD_CALIB".HMI_Manual_Pulse,
                         W_OUT => "PLC_DATA".RE_WSB,
                         X_OUT => "C#6_WD_CALIB".XUNG_SB1);
   END_IF;
   "C#6_WD_CALIB".KLT_AG1 := "PLC_DATA".RE_WAG;
   "C#6_WD_CALIB".KLT_FD1 := "PLC_DATA".RE_WFD;
   "C#6_WD_CALIB".KLT_AP1 := "PLC_DATA".RE_WAP;
   "C#6_WD_CALIB".KLT_SB1 := "PLC_DATA".RE_WSB;
   "1. CONVER TC"(AI := "AI_TEMP_TL",
                  HS := "C#6_WD_CALIB"."HS_TEMP TL",
                  TEMP_OUT => "PLC_DATA".TEMP_TL,
                  XUNG_OUT => "C#6_WD_CALIB".XUNG_TEMP_TL,
                  ENO => #_w4);
   "1. CONVER TC"(EN := #_w4,
                  AI := "AI_TEMP_TS",
                  HS := "C#6_WD_CALIB"."HS_TEMP TS",
                  TEMP_OUT => "PLC_DATA".TEMP_TS,
                  XUNG_OUT => "C#6_WD_CALIB".XUNG_TEMP_TS,
                  ENO => #_w5);
   "1. CONVER TC"(EN := #_w5,
                  AI := "AI_TEMP_AP",
                  HS := "C#6_WD_CALIB"."HS_TEMP AP",
                  TEMP_OUT => "PLC_DATA".TEMP_AP,
                  XUNG_OUT => "C#6_WD_CALIB".XUNG_TEMP_AP,
                  ENO => #_w6);
   IF #_w6 THEN
       "1. CONVER TC"(AI := "AI_TEMP_AG",
                      HS := "C#6_WD_CALIB"."HS_TEMP AG",
                      TEMP_OUT => "PLC_DATA".TEMP_AG,
                      XUNG_OUT => "C#6_WD_CALIB".XUNG_TEMP_AG);
   END_IF;
   "C#6_WD_CALIB".NDT_TL := DINT_TO_REAL("PLC_DATA".TEMP_TL);
   "C#6_WD_CALIB".NDT_TS := DINT_TO_REAL("PLC_DATA".TEMP_TS);
   "C#6_WD_CALIB".NDT_AP := DINT_TO_REAL("PLC_DATA".TEMP_AP);
   "C#6_WD_CALIB".NDT_AG := DINT_TO_REAL("PLC_DATA".TEMP_AG);
   "C#7_RD_RUN".TEMP_TUILOC := "PLC_DATA".TEMP_TL+0.0;
   "C#7_RD_RUN".TEMP_TANSAY := "PLC_DATA".TEMP_TS+0.0;
   "C#7_RD_RUN".TEMP_NHUA := "PLC_DATA".TEMP_AP+0.0;
   "C#7_RD_RUN".TEMP_AGG := "PLC_DATA".TEMP_AG+0.0;
END_REGION

REGION Network 5: CONVERT ANALOG IN PUT (0.0/ 0-10V: 1.0/4-20mA: 2.0/0-20mA) - Mode Độc Lập
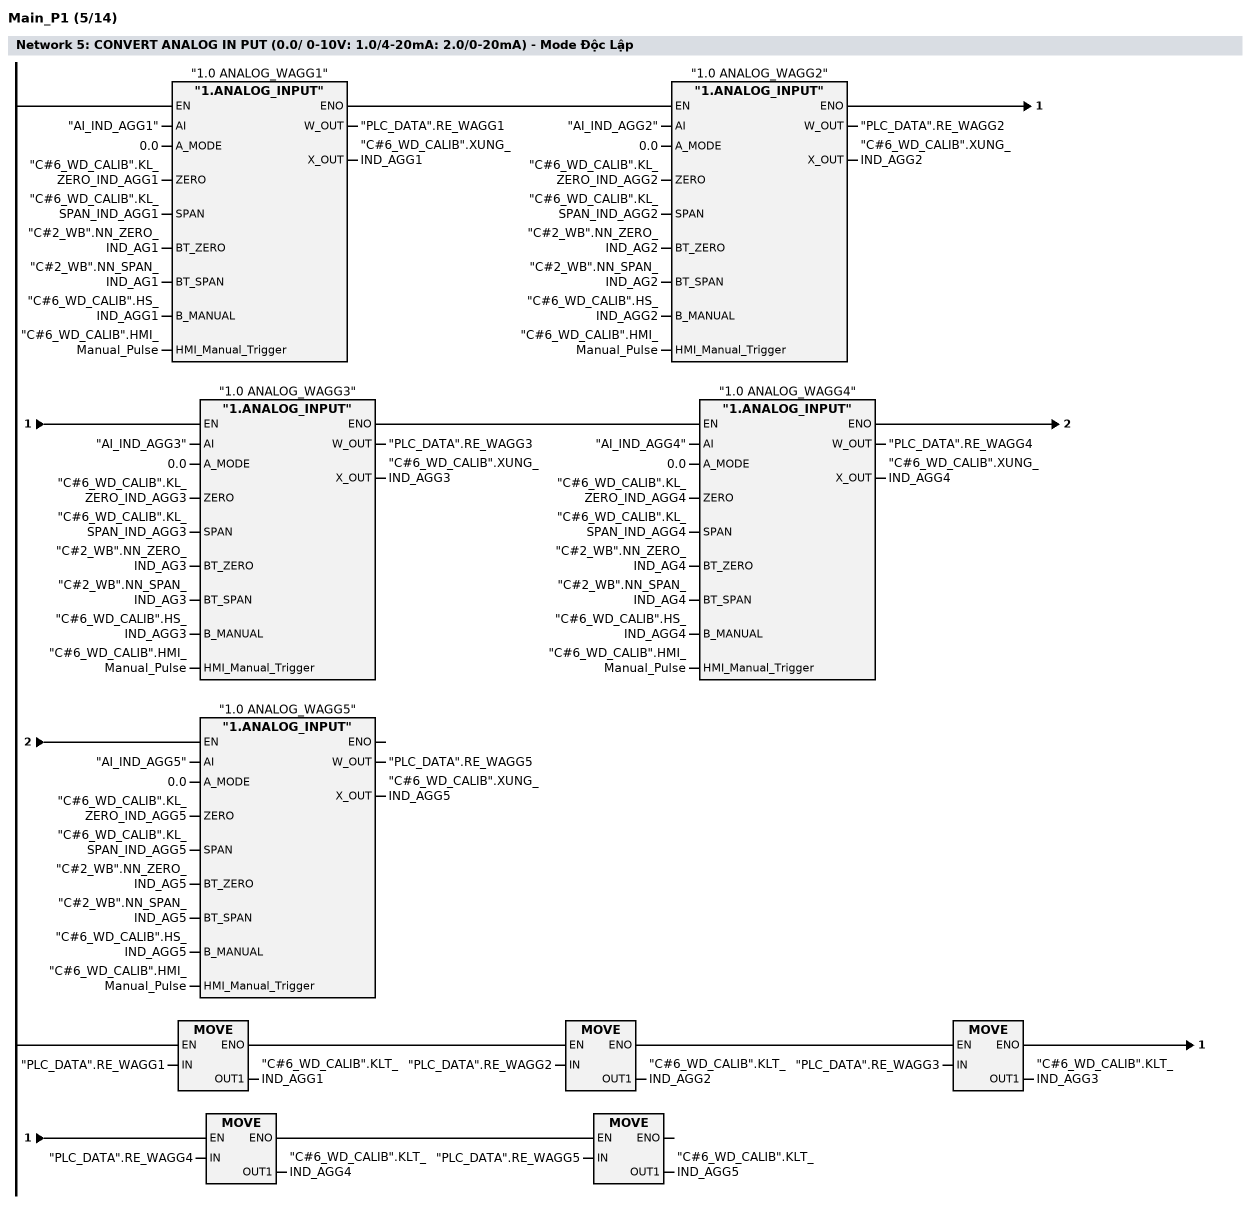
   RUNG wire#powerrail
      "1.0 ANALOG_WAGG1"(AI := "AI_IND_AGG1", A_MODE := 0.0, ZERO := "C#6_WD_CALIB".KL_ZERO_IND_AGG1, SPAN := "C#6_WD_CALIB".KL_SPAN_IND_AGG1, BT_ZERO := "C#2_WB".NN_ZERO_IND_AG1, BT_SPAN := "C#2_WB".NN_SPAN_IND_AG1, B_MANUAL := "C#6_WD_CALIB".HS_IND_AGG1, HMI_Manual_Trigger := "C#6_WD_CALIB".HMI_Manual_Pulse, W_OUT => "PLC_DATA".RE_WAGG1, X_OUT => "C#6_WD_CALIB".XUNG_IND_AGG1)
      "1.0 ANALOG_WAGG2"(AI := "AI_IND_AGG2", A_MODE := 0.0, ZERO := "C#6_WD_CALIB".KL_ZERO_IND_AGG2, SPAN := "C#6_WD_CALIB".KL_SPAN_IND_AGG2, BT_ZERO := "C#2_WB".NN_ZERO_IND_AG2, BT_SPAN := "C#2_WB".NN_SPAN_IND_AG2, B_MANUAL := "C#6_WD_CALIB".HS_IND_AGG2, HMI_Manual_Trigger := "C#6_WD_CALIB".HMI_Manual_Pulse, W_OUT => "PLC_DATA".RE_WAGG2, X_OUT => "C#6_WD_CALIB".XUNG_IND_AGG2)
      "1.0 ANALOG_WAGG3"(AI := "AI_IND_AGG3", A_MODE := 0.0, ZERO := "C#6_WD_CALIB".KL_ZERO_IND_AGG3, SPAN := "C#6_WD_CALIB".KL_SPAN_IND_AGG3, BT_ZERO := "C#2_WB".NN_ZERO_IND_AG3, BT_SPAN := "C#2_WB".NN_SPAN_IND_AG3, B_MANUAL := "C#6_WD_CALIB".HS_IND_AGG3, HMI_Manual_Trigger := "C#6_WD_CALIB".HMI_Manual_Pulse, W_OUT => "PLC_DATA".RE_WAGG3, X_OUT => "C#6_WD_CALIB".XUNG_IND_AGG3)
      "1.0 ANALOG_WAGG4"(AI := "AI_IND_AGG4", A_MODE := 0.0, ZERO := "C#6_WD_CALIB".KL_ZERO_IND_AGG4, SPAN := "C#6_WD_CALIB".KL_SPAN_IND_AGG4, BT_ZERO := "C#2_WB".NN_ZERO_IND_AG4, BT_SPAN := "C#2_WB".NN_SPAN_IND_AG4, B_MANUAL := "C#6_WD_CALIB".HS_IND_AGG4, HMI_Manual_Trigger := "C#6_WD_CALIB".HMI_Manual_Pulse, W_OUT => "PLC_DATA".RE_WAGG4, X_OUT => "C#6_WD_CALIB".XUNG_IND_AGG4)
      "1.0 ANALOG_WAGG5"(AI := "AI_IND_AGG5", A_MODE := 0.0, ZERO := "C#6_WD_CALIB".KL_ZERO_IND_AGG5, SPAN := "C#6_WD_CALIB".KL_SPAN_IND_AGG5, BT_ZERO := "C#2_WB".NN_ZERO_IND_AG5, BT_SPAN := "C#2_WB".NN_SPAN_IND_AG5, B_MANUAL := "C#6_WD_CALIB".HS_IND_AGG5, HMI_Manual_Trigger := "C#6_WD_CALIB".HMI_Manual_Pulse, W_OUT => "PLC_DATA".RE_WAGG5, X_OUT => "C#6_WD_CALIB".XUNG_IND_AGG5)
   END_RUNG
   RUNG wire#powerrail
      { S7_GenerateENO := "TRUE" } Move(in := "PLC_DATA".RE_WAGG1, out1 => "C#6_WD_CALIB".KLT_IND_AGG1)
      { S7_GenerateENO := "TRUE" } Move(in := "PLC_DATA".RE_WAGG2, out1 => "C#6_WD_CALIB".KLT_IND_AGG2)
      { S7_GenerateENO := "TRUE" } Move(in := "PLC_DATA".RE_WAGG3, out1 => "C#6_WD_CALIB".KLT_IND_AGG3)
      { S7_GenerateENO := "TRUE" } Move(in := "PLC_DATA".RE_WAGG4, out1 => "C#6_WD_CALIB".KLT_IND_AGG4)
      { S7_GenerateENO := "TRUE" } Move(in := "PLC_DATA".RE_WAGG5, out1 => "C#6_WD_CALIB".KLT_IND_AGG5)
   END_RUNG
   // the same network as SCL:
   // ENO of a box is taken as its EN; it also drops when the box reports an error
   "1.0 ANALOG_WAGG1"(AI := "AI_IND_AGG1",   // "1.ANALOG_INPUT"
                      A_MODE := 0.0,
                      ZERO := "C#6_WD_CALIB".KL_ZERO_IND_AGG1,
                      SPAN := "C#6_WD_CALIB".KL_SPAN_IND_AGG1,
                      BT_ZERO := "C#2_WB".NN_ZERO_IND_AG1,
                      BT_SPAN := "C#2_WB".NN_SPAN_IND_AG1,
                      B_MANUAL := "C#6_WD_CALIB".HS_IND_AGG1,
                      HMI_Manual_Trigger := "C#6_WD_CALIB".HMI_Manual_Pulse,
                      W_OUT => "PLC_DATA".RE_WAGG1,
                      X_OUT => "C#6_WD_CALIB".XUNG_IND_AGG1,
                      ENO => #_w1);
   "1.0 ANALOG_WAGG2"(EN := #_w1,   // "1.ANALOG_INPUT"
                      AI := "AI_IND_AGG2",
                      A_MODE := 0.0,
                      ZERO := "C#6_WD_CALIB".KL_ZERO_IND_AGG2,
                      SPAN := "C#6_WD_CALIB".KL_SPAN_IND_AGG2,
                      BT_ZERO := "C#2_WB".NN_ZERO_IND_AG2,
                      BT_SPAN := "C#2_WB".NN_SPAN_IND_AG2,
                      B_MANUAL := "C#6_WD_CALIB".HS_IND_AGG2,
                      HMI_Manual_Trigger := "C#6_WD_CALIB".HMI_Manual_Pulse,
                      W_OUT => "PLC_DATA".RE_WAGG2,
                      X_OUT => "C#6_WD_CALIB".XUNG_IND_AGG2,
                      ENO => #_w2);
   "1.0 ANALOG_WAGG3"(EN := #_w2,   // "1.ANALOG_INPUT"
                      AI := "AI_IND_AGG3",
                      A_MODE := 0.0,
                      ZERO := "C#6_WD_CALIB".KL_ZERO_IND_AGG3,
                      SPAN := "C#6_WD_CALIB".KL_SPAN_IND_AGG3,
                      BT_ZERO := "C#2_WB".NN_ZERO_IND_AG3,
                      BT_SPAN := "C#2_WB".NN_SPAN_IND_AG3,
                      B_MANUAL := "C#6_WD_CALIB".HS_IND_AGG3,
                      HMI_Manual_Trigger := "C#6_WD_CALIB".HMI_Manual_Pulse,
                      W_OUT => "PLC_DATA".RE_WAGG3,
                      X_OUT => "C#6_WD_CALIB".XUNG_IND_AGG3,
                      ENO => #_w3);
   "1.0 ANALOG_WAGG4"(EN := #_w3,   // "1.ANALOG_INPUT"
                      AI := "AI_IND_AGG4",
                      A_MODE := 0.0,
                      ZERO := "C#6_WD_CALIB".KL_ZERO_IND_AGG4,
                      SPAN := "C#6_WD_CALIB".KL_SPAN_IND_AGG4,
                      BT_ZERO := "C#2_WB".NN_ZERO_IND_AG4,
                      BT_SPAN := "C#2_WB".NN_SPAN_IND_AG4,
                      B_MANUAL := "C#6_WD_CALIB".HS_IND_AGG4,
                      HMI_Manual_Trigger := "C#6_WD_CALIB".HMI_Manual_Pulse,
                      W_OUT => "PLC_DATA".RE_WAGG4,
                      X_OUT => "C#6_WD_CALIB".XUNG_IND_AGG4,
                      ENO => #_w4);
   IF #_w4 THEN
       "1.0 ANALOG_WAGG5"(AI := "AI_IND_AGG5",   // "1.ANALOG_INPUT"
                          A_MODE := 0.0,
                          ZERO := "C#6_WD_CALIB".KL_ZERO_IND_AGG5,
                          SPAN := "C#6_WD_CALIB".KL_SPAN_IND_AGG5,
                          BT_ZERO := "C#2_WB".NN_ZERO_IND_AG5,
                          BT_SPAN := "C#2_WB".NN_SPAN_IND_AG5,
                          B_MANUAL := "C#6_WD_CALIB".HS_IND_AGG5,
                          HMI_Manual_Trigger := "C#6_WD_CALIB".HMI_Manual_Pulse,
                          W_OUT => "PLC_DATA".RE_WAGG5,
                          X_OUT => "C#6_WD_CALIB".XUNG_IND_AGG5);
   END_IF;
   "C#6_WD_CALIB".KLT_IND_AGG1 := "PLC_DATA".RE_WAGG1;
   "C#6_WD_CALIB".KLT_IND_AGG2 := "PLC_DATA".RE_WAGG2;
   "C#6_WD_CALIB".KLT_IND_AGG3 := "PLC_DATA".RE_WAGG3;
   "C#6_WD_CALIB".KLT_IND_AGG4 := "PLC_DATA".RE_WAGG4;
   "C#6_WD_CALIB".KLT_IND_AGG5 := "PLC_DATA".RE_WAGG5;
END_REGION

REGION Network 6: RUN MODE
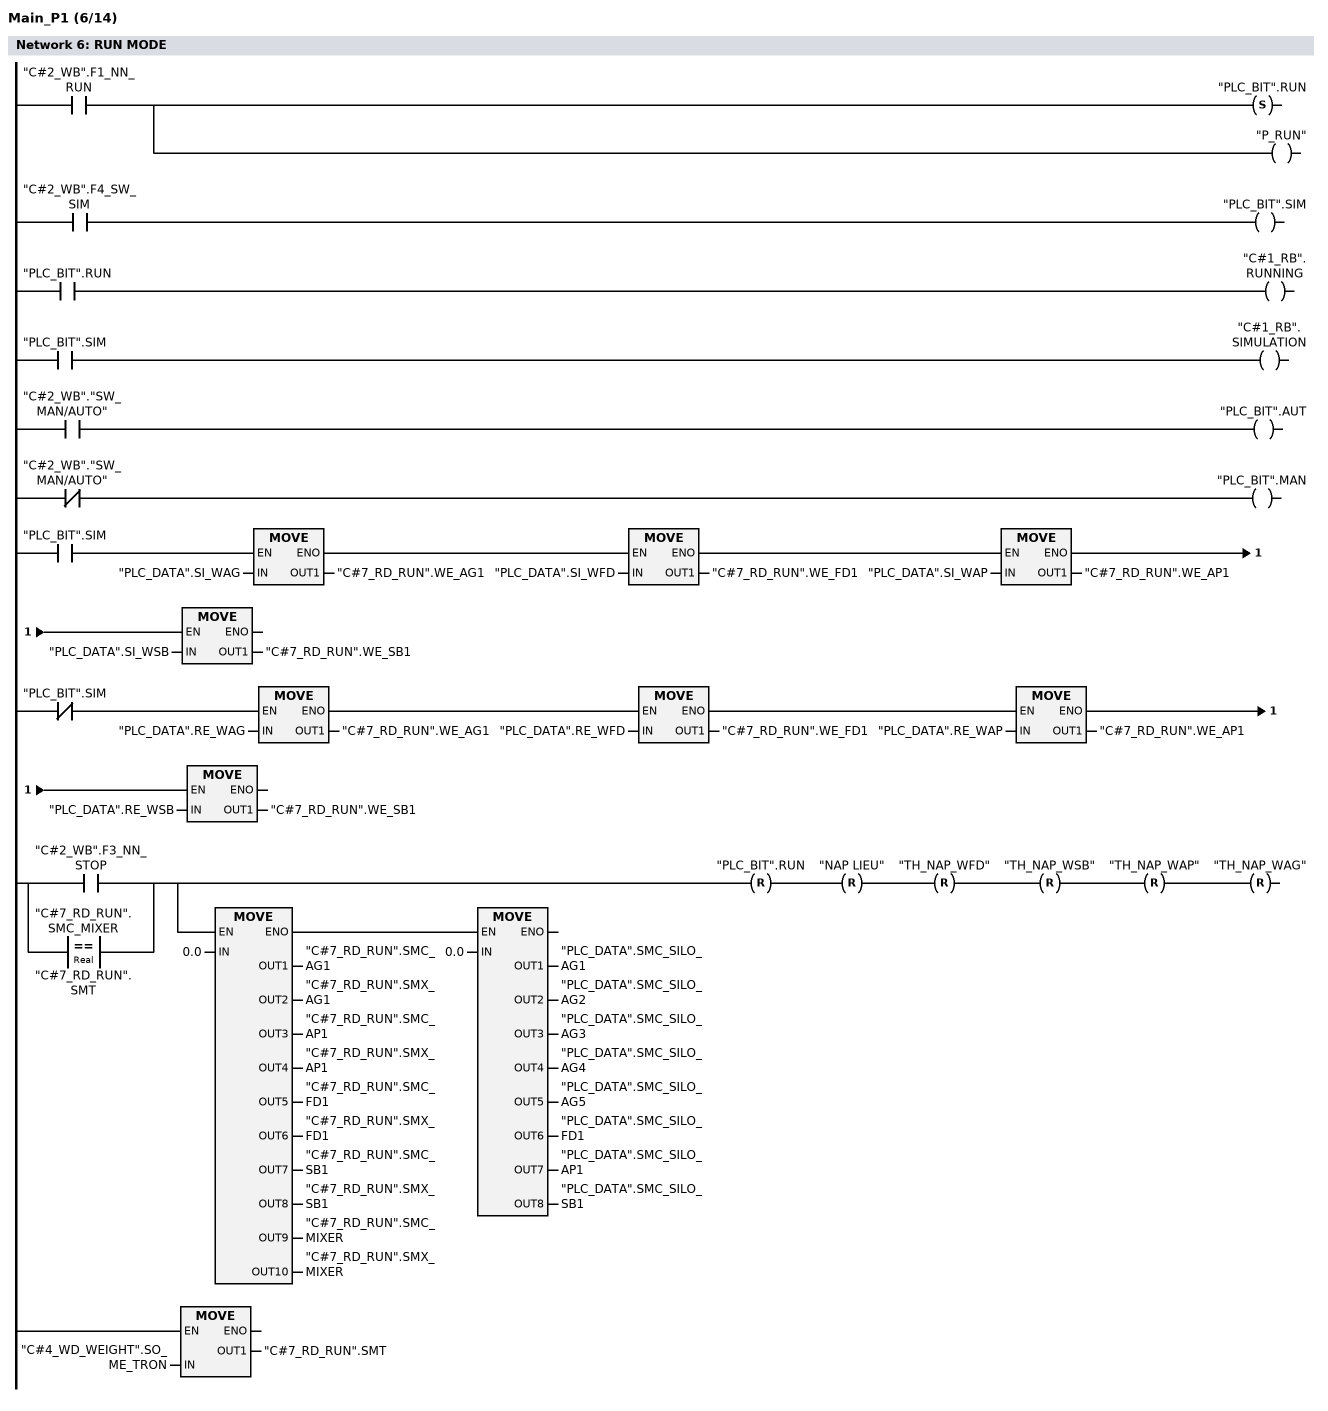
   RUNG wire#powerrail
      Contact( "C#2_WB".F1_NN_RUN )
      wire#w1
      S_Coil( "PLC_BIT".RUN )
   END_RUNG
   RUNG wire#w1
      Coil( "P_RUN" )
   END_RUNG
   RUNG wire#powerrail
      Contact( "C#2_WB".F4_SW_SIM )
      Coil( "PLC_BIT".SIM )
   END_RUNG
   RUNG wire#powerrail
      Contact( "PLC_BIT".RUN )
      Coil( "C#1_RB".RUNNING )
   END_RUNG
   RUNG wire#powerrail
      Contact( "PLC_BIT".SIM )
      Coil( "C#1_RB".SIMULATION )
   END_RUNG
   RUNG wire#powerrail
      Contact( "C#2_WB"."SW_MAN/AUTO" )
      Coil( "PLC_BIT".AUT )
   END_RUNG
   RUNG wire#powerrail
      I_Contact( "C#2_WB"."SW_MAN/AUTO" )
      Coil( "PLC_BIT".MAN )
   END_RUNG
   RUNG wire#powerrail
      Contact( "PLC_BIT".SIM )
      { S7_GenerateENO := "TRUE" } Move(in := "PLC_DATA".SI_WAG, out1 => "C#7_RD_RUN".WE_AG1)
      { S7_GenerateENO := "TRUE" } Move(in := "PLC_DATA".SI_WFD, out1 => "C#7_RD_RUN".WE_FD1)
      { S7_GenerateENO := "TRUE" } Move(in := "PLC_DATA".SI_WAP, out1 => "C#7_RD_RUN".WE_AP1)
      { S7_GenerateENO := "TRUE" } Move(in := "PLC_DATA".SI_WSB, out1 => "C#7_RD_RUN".WE_SB1)
   END_RUNG
   RUNG wire#powerrail
      I_Contact( "PLC_BIT".SIM )
      { S7_GenerateENO := "TRUE" } Move(in := "PLC_DATA".RE_WAG, out1 => "C#7_RD_RUN".WE_AG1)
      { S7_GenerateENO := "TRUE" } Move(in := "PLC_DATA".RE_WFD, out1 => "C#7_RD_RUN".WE_FD1)
      { S7_GenerateENO := "TRUE" } Move(in := "PLC_DATA".RE_WAP, out1 => "C#7_RD_RUN".WE_AP1)
      { S7_GenerateENO := "TRUE" } Move(in := "PLC_DATA".RE_WSB, out1 => "C#7_RD_RUN".WE_SB1)
   END_RUNG
   RUNG wire#powerrail
      Contact( "C#2_WB".F3_NN_STOP )
      wire#w2
      R_Coil( "PLC_BIT".RUN )
      R_Coil( "NAP LIEU" )
      R_Coil( "TH_NAP_WFD" )
      R_Coil( "TH_NAP_WSB" )
      R_Coil( "TH_NAP_WAP" )
      R_Coil( "TH_NAP_WAG" )
   END_RUNG
   RUNG wire#powerrail
      { S7_Templates := "SrcType := Real" } EQ_Contact(in1 := "C#7_RD_RUN".SMC_MIXER, in2 := "C#7_RD_RUN".SMT)
   END_RUNG wire#w2
   RUNG wire#w2
      { S7_GenerateENO := "TRUE" } Move(in := 0.0, out1 => "C#7_RD_RUN".SMC_AG1, out2 => "C#7_RD_RUN".SMX_AG1, out3 => "C#7_RD_RUN".SMC_AP1, out4 => "C#7_RD_RUN".SMX_AP1, out5 => "C#7_RD_RUN".SMC_FD1, out6 => "C#7_RD_RUN".SMX_FD1, out7 => "C#7_RD_RUN".SMC_SB1, out8 => "C#7_RD_RUN".SMX_SB1, out9 => "C#7_RD_RUN".SMC_MIXER, out10 => "C#7_RD_RUN".SMX_MIXER)
      { S7_GenerateENO := "TRUE" } Move(in := 0.0, out1 => "PLC_DATA".SMC_SILO_AG1, out2 => "PLC_DATA".SMC_SILO_AG2, out3 => "PLC_DATA".SMC_SILO_AG3, out4 => "PLC_DATA".SMC_SILO_AG4, out5 => "PLC_DATA".SMC_SILO_AG5, out6 => "PLC_DATA".SMC_SILO_FD1, out7 => "PLC_DATA".SMC_SILO_AP1, out8 => "PLC_DATA".SMC_SILO_SB1)
   END_RUNG
   RUNG wire#powerrail
      Move(in := "C#4_WD_WEIGHT".SO_ME_TRON, out1 => "C#7_RD_RUN".SMT)
   END_RUNG
   // the same network as SCL:
   // ENO of a box is taken as its EN; it also drops when the box reports an error
   IF "C#2_WB".F1_NN_RUN THEN "PLC_BIT".RUN := TRUE; END_IF;
   "P_RUN" := "C#2_WB".F1_NN_RUN;
   "PLC_BIT".SIM := "C#2_WB".F4_SW_SIM;
   "C#1_RB".RUNNING := "PLC_BIT".RUN;
   "C#1_RB".SIMULATION := "PLC_BIT".SIM;
   "PLC_BIT".AUT := "C#2_WB"."SW_MAN/AUTO";
   "PLC_BIT".MAN := NOT "C#2_WB"."SW_MAN/AUTO";
   IF "PLC_BIT".SIM THEN
       "C#7_RD_RUN".WE_AG1 := "PLC_DATA".SI_WAG;
       "C#7_RD_RUN".WE_FD1 := "PLC_DATA".SI_WFD;
       "C#7_RD_RUN".WE_AP1 := "PLC_DATA".SI_WAP;
       "C#7_RD_RUN".WE_SB1 := "PLC_DATA".SI_WSB;
   END_IF;
   IF NOT "PLC_BIT".SIM THEN
       "C#7_RD_RUN".WE_AG1 := "PLC_DATA".RE_WAG;
       "C#7_RD_RUN".WE_FD1 := "PLC_DATA".RE_WFD;
       "C#7_RD_RUN".WE_AP1 := "PLC_DATA".RE_WAP;
       "C#7_RD_RUN".WE_SB1 := "PLC_DATA".RE_WSB;
   END_IF;
   IF "C#2_WB".F3_NN_STOP OR ("C#7_RD_RUN".SMC_MIXER = "C#7_RD_RUN".SMT) THEN
       "PLC_BIT".RUN := FALSE;
       "NAP LIEU" := FALSE;
       "TH_NAP_WFD" := FALSE;
       "TH_NAP_WSB" := FALSE;
       "TH_NAP_WAP" := FALSE;
       "TH_NAP_WAG" := FALSE;
   END_IF;
   #_w1 := "C#2_WB".F3_NN_STOP OR ("C#7_RD_RUN".SMC_MIXER = "C#7_RD_RUN".SMT);
   IF #_w1 THEN
       "C#7_RD_RUN".SMC_AG1 := 0.0;
       "C#7_RD_RUN".SMX_AG1 := 0.0;
       "C#7_RD_RUN".SMC_AP1 := 0.0;
       "C#7_RD_RUN".SMX_AP1 := 0.0;
       "C#7_RD_RUN".SMC_FD1 := 0.0;
       "C#7_RD_RUN".SMX_FD1 := 0.0;
       "C#7_RD_RUN".SMC_SB1 := 0.0;
       "C#7_RD_RUN".SMX_SB1 := 0.0;
       "C#7_RD_RUN".SMC_MIXER := 0.0;
       "C#7_RD_RUN".SMX_MIXER := 0.0;
       "PLC_DATA".SMC_SILO_AG1 := 0.0;
       "PLC_DATA".SMC_SILO_AG2 := 0.0;
       "PLC_DATA".SMC_SILO_AG3 := 0.0;
       "PLC_DATA".SMC_SILO_AG4 := 0.0;
       "PLC_DATA".SMC_SILO_AG5 := 0.0;
       "PLC_DATA".SMC_SILO_FD1 := 0.0;
       "PLC_DATA".SMC_SILO_AP1 := 0.0;
       "PLC_DATA".SMC_SILO_SB1 := 0.0;
   END_IF;
   "C#7_RD_RUN".SMT := "C#4_WD_WEIGHT".SO_ME_TRON;
END_REGION

REGION Network 7: DATA SIMULATION
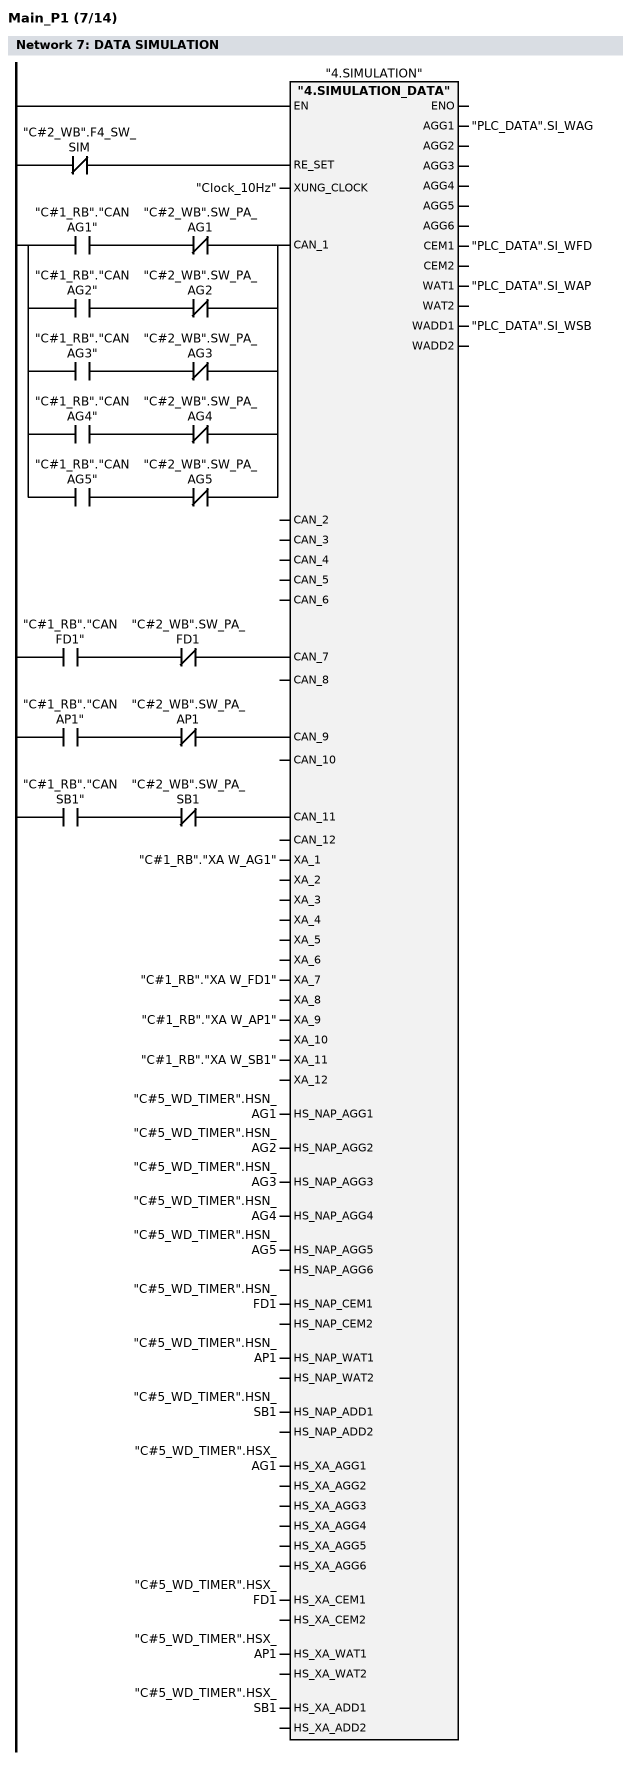
   RUNG wire#powerrail
      "4.SIMULATION"(RE_SET := wire#w1, CAN_1 := wire#w2, CAN_7 := wire#w3, CAN_9 := wire#w4, CAN_11 := wire#w5, XUNG_CLOCK := "Clock_10Hz", CAN_2 :=, CAN_3 :=, CAN_4 :=, CAN_5 :=, CAN_6 :=, CAN_8 :=, CAN_10 :=, CAN_12 :=, XA_1 := "C#1_RB"."XA W_AG1", XA_2 :=, XA_3 :=, XA_4 :=, XA_5 :=, XA_6 :=, XA_7 := "C#1_RB"."XA W_FD1", XA_8 :=, XA_9 := "C#1_RB"."XA W_AP1", XA_10 :=, XA_11 := "C#1_RB"."XA W_SB1", XA_12 :=, HS_NAP_AGG1 := "C#5_WD_TIMER".HSN_AG1, HS_NAP_AGG2 := "C#5_WD_TIMER".HSN_AG2, HS_NAP_AGG3 := "C#5_WD_TIMER".HSN_AG3, HS_NAP_AGG4 := "C#5_WD_TIMER".HSN_AG4, HS_NAP_AGG5 := "C#5_WD_TIMER".HSN_AG5, HS_NAP_AGG6 :=, HS_NAP_CEM1 := "C#5_WD_TIMER".HSN_FD1, HS_NAP_CEM2 :=, HS_NAP_WAT1 := "C#5_WD_TIMER".HSN_AP1, HS_NAP_WAT2 :=, HS_NAP_ADD1 := "C#5_WD_TIMER".HSN_SB1, HS_NAP_ADD2 :=, HS_XA_AGG1 := "C#5_WD_TIMER".HSX_AG1, HS_XA_AGG2 :=, HS_XA_AGG3 :=, HS_XA_AGG4 :=, HS_XA_AGG5 :=, HS_XA_AGG6 :=, HS_XA_CEM1 := "C#5_WD_TIMER".HSX_FD1, HS_XA_CEM2 :=, HS_XA_WAT1 := "C#5_WD_TIMER".HSX_AP1, HS_XA_WAT2 :=, HS_XA_ADD1 := "C#5_WD_TIMER".HSX_SB1, HS_XA_ADD2 :=, AGG1 => "PLC_DATA".SI_WAG, AGG2 =>, AGG3 =>, AGG4 =>, AGG5 =>, AGG6 =>, CEM1 => "PLC_DATA".SI_WFD, CEM2 =>, WAT1 => "PLC_DATA".SI_WAP, WAT2 =>, WADD1 => "PLC_DATA".SI_WSB, WADD2 =>)
   END_RUNG
   RUNG wire#powerrail
      I_Contact( "C#2_WB".F4_SW_SIM )
   END_RUNG wire#w1
   RUNG wire#powerrail
      Contact( "C#1_RB"."CAN AG1" )
      I_Contact( "C#2_WB".SW_PA_AG1 )
   END_RUNG wire#w2
   RUNG wire#powerrail
      Contact( "C#1_RB"."CAN AG2" )
      I_Contact( "C#2_WB".SW_PA_AG2 )
   END_RUNG wire#w2
   RUNG wire#powerrail
      Contact( "C#1_RB"."CAN AG3" )
      I_Contact( "C#2_WB".SW_PA_AG3 )
   END_RUNG wire#w2
   RUNG wire#powerrail
      Contact( "C#1_RB"."CAN AG4" )
      I_Contact( "C#2_WB".SW_PA_AG4 )
   END_RUNG wire#w2
   RUNG wire#powerrail
      Contact( "C#1_RB"."CAN AG5" )
      I_Contact( "C#2_WB".SW_PA_AG5 )
   END_RUNG wire#w2
   RUNG wire#powerrail
      Contact( "C#1_RB"."CAN FD1" )
      I_Contact( "C#2_WB".SW_PA_FD1 )
   END_RUNG wire#w3
   RUNG wire#powerrail
      Contact( "C#1_RB"."CAN AP1" )
      I_Contact( "C#2_WB".SW_PA_AP1 )
   END_RUNG wire#w4
   RUNG wire#powerrail
      Contact( "C#1_RB"."CAN SB1" )
      I_Contact( "C#2_WB".SW_PA_SB1 )
   END_RUNG wire#w5
   // the same network as SCL:
   "4.SIMULATION"(RE_SET := NOT "C#2_WB".F4_SW_SIM,   // "4.SIMULATION_DATA"
                  XUNG_CLOCK := "Clock_10Hz",
                  CAN_1 := ("C#1_RB"."CAN AG1" AND NOT "C#2_WB".SW_PA_AG1) OR ("C#1_RB"."CAN AG2" AND NOT "C#2_WB".SW_PA_AG2) OR ("C#1_RB"."CAN AG3" AND NOT "C#2_WB".SW_PA_AG3) OR ("C#1_RB"."CAN AG4" AND NOT "C#2_WB".SW_PA_AG4) OR ("C#1_RB"."CAN AG5" AND NOT "C#2_WB".SW_PA_AG5),
                  CAN_7 := "C#1_RB"."CAN FD1" AND NOT "C#2_WB".SW_PA_FD1,
                  CAN_9 := "C#1_RB"."CAN AP1" AND NOT "C#2_WB".SW_PA_AP1,
                  CAN_11 := "C#1_RB"."CAN SB1" AND NOT "C#2_WB".SW_PA_SB1,
                  XA_1 := "C#1_RB"."XA W_AG1",
                  XA_7 := "C#1_RB"."XA W_FD1",
                  XA_9 := "C#1_RB"."XA W_AP1",
                  XA_11 := "C#1_RB"."XA W_SB1",
                  HS_NAP_AGG1 := "C#5_WD_TIMER".HSN_AG1,
                  HS_NAP_AGG2 := "C#5_WD_TIMER".HSN_AG2,
                  HS_NAP_AGG3 := "C#5_WD_TIMER".HSN_AG3,
                  HS_NAP_AGG4 := "C#5_WD_TIMER".HSN_AG4,
                  HS_NAP_AGG5 := "C#5_WD_TIMER".HSN_AG5,
                  HS_NAP_CEM1 := "C#5_WD_TIMER".HSN_FD1,
                  HS_NAP_WAT1 := "C#5_WD_TIMER".HSN_AP1,
                  HS_NAP_ADD1 := "C#5_WD_TIMER".HSN_SB1,
                  HS_XA_AGG1 := "C#5_WD_TIMER".HSX_AG1,
                  HS_XA_CEM1 := "C#5_WD_TIMER".HSX_FD1,
                  HS_XA_WAT1 := "C#5_WD_TIMER".HSX_AP1,
                  HS_XA_ADD1 := "C#5_WD_TIMER".HSX_SB1,
                  AGG1 => "PLC_DATA".SI_WAG,
                  CEM1 => "PLC_DATA".SI_WFD,
                  WAT1 => "PLC_DATA".SI_WAP,
                  WADD1 => "PLC_DATA".SI_WSB);
END_REGION

REGION Network 8: XỬ LÍ CÂN CỐT LIỆU
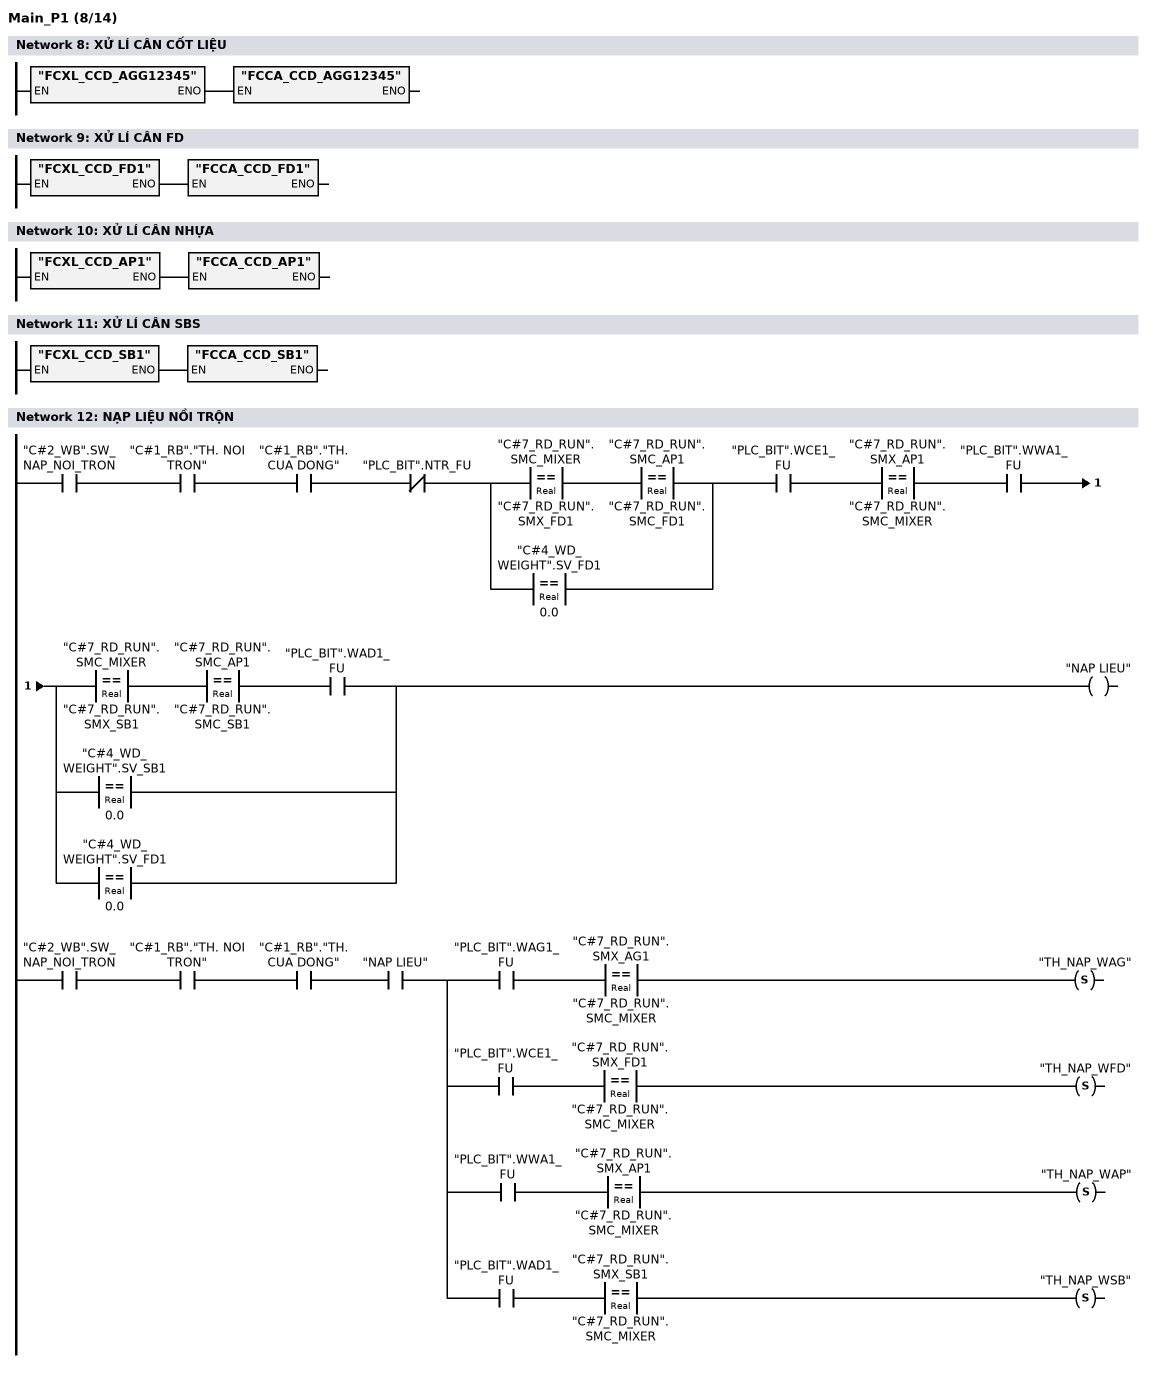
   RUNG wire#powerrail
      "FCXL_CCD_AGG12345"()
      "FCCA_CCD_AGG12345"()
   END_RUNG
   // the same network as SCL:
   "FCXL_CCD_AGG12345"(ENO => #_w1);
   IF #_w1 THEN "FCCA_CCD_AGG12345"(); END_IF;
END_REGION

REGION Network 9: XỬ LÍ CÂN FD
   RUNG wire#powerrail
      "FCXL_CCD_FD1"()
      "FCCA_CCD_FD1"()
   END_RUNG
   // the same network as SCL:
   "FCXL_CCD_FD1"(ENO => #_w1);
   IF #_w1 THEN "FCCA_CCD_FD1"(); END_IF;
END_REGION

REGION Network 10: XỬ LÍ CÂN NHỰA
   RUNG wire#powerrail
      "FCXL_CCD_AP1"()
      "FCCA_CCD_AP1"()
   END_RUNG
   // the same network as SCL:
   "FCXL_CCD_AP1"(ENO => #_w1);
   IF #_w1 THEN "FCCA_CCD_AP1"(); END_IF;
END_REGION

REGION Network 11: XỬ LÍ CÂN SBS
   RUNG wire#powerrail
      "FCXL_CCD_SB1"()
      "FCCA_CCD_SB1"()
   END_RUNG
   // the same network as SCL:
   "FCXL_CCD_SB1"(ENO => #_w1);
   IF #_w1 THEN "FCCA_CCD_SB1"(); END_IF;
END_REGION

REGION Network 12: NẠP LIỆU NỒI TRỘN
   RUNG wire#powerrail
      Contact( "C#2_WB".SW_NAP_NOI_TRON )
      Contact( "C#1_RB"."TH. NOI TRON" )
      Contact( "C#1_RB"."TH. CUA DONG" )
      I_Contact( "PLC_BIT".NTR_FU )
      wire#w1
      { S7_Templates := "SrcType := Real" } EQ_Contact(in1 := "C#7_RD_RUN".SMC_MIXER, in2 := "C#7_RD_RUN".SMX_FD1)
      { S7_Templates := "SrcType := Real" } EQ_Contact(in1 := "C#7_RD_RUN".SMC_AP1, in2 := "C#7_RD_RUN".SMC_FD1)
      wire#w2
      Contact( "PLC_BIT".WCE1_FU )
      { S7_Templates := "SrcType := Real" } EQ_Contact(in1 := "C#7_RD_RUN".SMX_AP1, in2 := "C#7_RD_RUN".SMC_MIXER)
      Contact( "PLC_BIT".WWA1_FU )
      wire#w3
      { S7_Templates := "SrcType := Real" } EQ_Contact(in1 := "C#7_RD_RUN".SMC_MIXER, in2 := "C#7_RD_RUN".SMX_SB1)
      { S7_Templates := "SrcType := Real" } EQ_Contact(in1 := "C#7_RD_RUN".SMC_AP1, in2 := "C#7_RD_RUN".SMC_SB1)
      Contact( "PLC_BIT".WAD1_FU )
      wire#w4
      Coil( "NAP LIEU" )
   END_RUNG
   RUNG wire#w1
      { S7_Templates := "SrcType := Real" } EQ_Contact(in1 := "C#4_WD_WEIGHT".SV_FD1, in2 := 0.0)
   END_RUNG wire#w2
   RUNG wire#w3
      { S7_Templates := "SrcType := Real" } EQ_Contact(in1 := "C#4_WD_WEIGHT".SV_SB1, in2 := 0.0)
   END_RUNG wire#w4
   RUNG wire#w3
      { S7_Templates := "SrcType := Real" } EQ_Contact(in1 := "C#4_WD_WEIGHT".SV_FD1, in2 := 0.0)
   END_RUNG wire#w4
   RUNG wire#powerrail
      Contact( "C#2_WB".SW_NAP_NOI_TRON )
      Contact( "C#1_RB"."TH. NOI TRON" )
      Contact( "C#1_RB"."TH. CUA DONG" )
      Contact( "NAP LIEU" )
      wire#w5
      Contact( "PLC_BIT".WAG1_FU )
      { S7_Templates := "SrcType := Real" } EQ_Contact(in1 := "C#7_RD_RUN".SMX_AG1, in2 := "C#7_RD_RUN".SMC_MIXER)
      S_Coil( "TH_NAP_WAG" )
   END_RUNG
   RUNG wire#w5
      Contact( "PLC_BIT".WCE1_FU )
      { S7_Templates := "SrcType := Real" } EQ_Contact(in1 := "C#7_RD_RUN".SMX_FD1, in2 := "C#7_RD_RUN".SMC_MIXER)
      S_Coil( "TH_NAP_WFD" )
   END_RUNG
   RUNG wire#w5
      Contact( "PLC_BIT".WWA1_FU )
      { S7_Templates := "SrcType := Real" } EQ_Contact(in1 := "C#7_RD_RUN".SMX_AP1, in2 := "C#7_RD_RUN".SMC_MIXER)
      S_Coil( "TH_NAP_WAP" )
   END_RUNG
   RUNG wire#w5
      Contact( "PLC_BIT".WAD1_FU )
      { S7_Templates := "SrcType := Real" } EQ_Contact(in1 := "C#7_RD_RUN".SMX_SB1, in2 := "C#7_RD_RUN".SMC_MIXER)
      S_Coil( "TH_NAP_WSB" )
   END_RUNG
   // the same network as SCL:
   "NAP LIEU" := "C#2_WB".SW_NAP_NOI_TRON AND "C#1_RB"."TH. NOI TRON" AND "C#1_RB"."TH. CUA DONG" AND NOT "PLC_BIT".NTR_FU AND ((("C#7_RD_RUN".SMC_MIXER = "C#7_RD_RUN".SMX_FD1) AND ("C#7_RD_RUN".SMC_AP1 = "C#7_RD_RUN".SMC_FD1)) OR ("C#4_WD_WEIGHT".SV_FD1 = 0.0)) AND "PLC_BIT".WCE1_FU AND ("C#7_RD_RUN".SMX_AP1 = "C#7_RD_RUN".SMC_MIXER) AND "PLC_BIT".WWA1_FU AND ((("C#7_RD_RUN".SMC_MIXER = "C#7_RD_RUN".SMX_SB1) AND ("C#7_RD_RUN".SMC_AP1 = "C#7_RD_RUN".SMC_SB1) AND "PLC_BIT".WAD1_FU) OR ("C#4_WD_WEIGHT".SV_SB1 = 0.0) OR ("C#4_WD_WEIGHT".SV_FD1 = 0.0));
   #_w1 := "C#2_WB".SW_NAP_NOI_TRON AND "C#1_RB"."TH. NOI TRON" AND "C#1_RB"."TH. CUA DONG" AND "NAP LIEU";
   IF #_w1 AND "PLC_BIT".WAG1_FU AND ("C#7_RD_RUN".SMX_AG1 = "C#7_RD_RUN".SMC_MIXER) THEN
       "TH_NAP_WAG" := TRUE;
   END_IF;
   IF #_w1 AND "PLC_BIT".WCE1_FU AND ("C#7_RD_RUN".SMX_FD1 = "C#7_RD_RUN".SMC_MIXER) THEN
       "TH_NAP_WFD" := TRUE;
   END_IF;
   IF #_w1 AND "PLC_BIT".WWA1_FU AND ("C#7_RD_RUN".SMX_AP1 = "C#7_RD_RUN".SMC_MIXER) THEN
       "TH_NAP_WAP" := TRUE;
   END_IF;
   IF #_w1 AND "PLC_BIT".WAD1_FU AND ("C#7_RD_RUN".SMX_SB1 = "C#7_RD_RUN".SMC_MIXER) THEN
       "TH_NAP_WSB" := TRUE;
   END_IF;
END_REGION

REGION Network 13: XỬ LÍ NỒI TRỘN
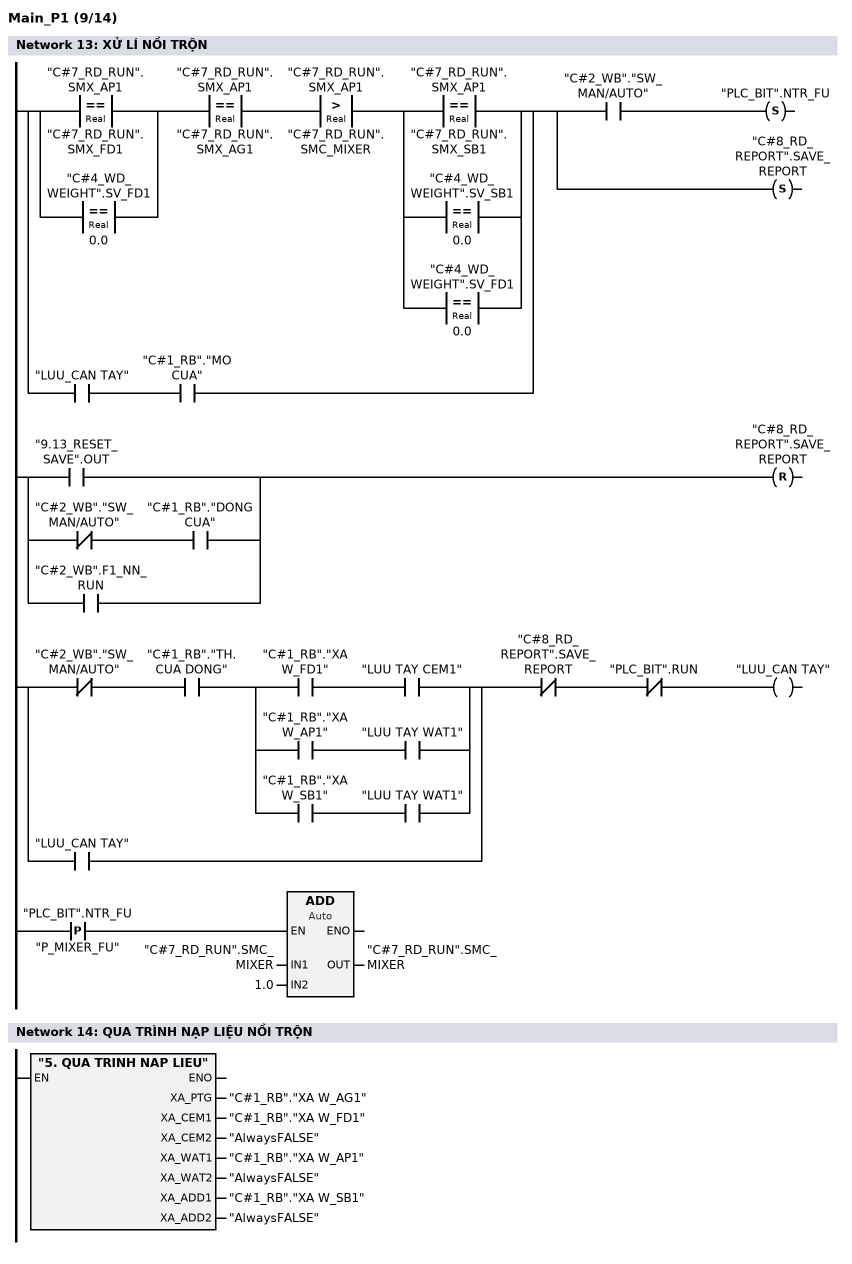
   RUNG wire#powerrail
      { S7_Templates := "SrcType := Real" } EQ_Contact(in1 := "C#7_RD_RUN".SMX_AP1, in2 := "C#7_RD_RUN".SMX_FD1)
      wire#w1
      { S7_Templates := "SrcType := Real" } EQ_Contact(in1 := "C#7_RD_RUN".SMX_AP1, in2 := "C#7_RD_RUN".SMX_AG1)
      { S7_Templates := "SrcType := Real" } GT_Contact(in1 := "C#7_RD_RUN".SMX_AP1, in2 := "C#7_RD_RUN".SMC_MIXER)
      wire#w2
      { S7_Templates := "SrcType := Real" } EQ_Contact(in1 := "C#7_RD_RUN".SMX_AP1, in2 := "C#7_RD_RUN".SMX_SB1)
      wire#w3
      Contact( "C#2_WB"."SW_MAN/AUTO" )
      S_Coil( "PLC_BIT".NTR_FU )
   END_RUNG
   RUNG wire#powerrail
      { S7_Templates := "SrcType := Real" } EQ_Contact(in1 := "C#4_WD_WEIGHT".SV_FD1, in2 := 0.0)
   END_RUNG wire#w1
   RUNG wire#w2
      { S7_Templates := "SrcType := Real" } EQ_Contact(in1 := "C#4_WD_WEIGHT".SV_SB1, in2 := 0.0)
   END_RUNG wire#w3
   RUNG wire#w2
      { S7_Templates := "SrcType := Real" } EQ_Contact(in1 := "C#4_WD_WEIGHT".SV_FD1, in2 := 0.0)
   END_RUNG wire#w3
   RUNG wire#powerrail
      Contact( "LUU_CAN TAY" )
      Contact( "C#1_RB"."MO CUA" )
   END_RUNG wire#w3
   RUNG wire#w3
      S_Coil( "C#8_RD_REPORT".SAVE_REPORT )
   END_RUNG
   RUNG wire#powerrail
      Contact( "9.13_RESET_SAVE".OUT )
      wire#w4
      R_Coil( "C#8_RD_REPORT".SAVE_REPORT )
   END_RUNG
   RUNG wire#powerrail
      I_Contact( "C#2_WB"."SW_MAN/AUTO" )
      Contact( "C#1_RB"."DONG CUA" )
   END_RUNG wire#w4
   RUNG wire#powerrail
      Contact( "C#2_WB".F1_NN_RUN )
   END_RUNG wire#w4
   RUNG wire#powerrail
      I_Contact( "C#2_WB"."SW_MAN/AUTO" )
      Contact( "C#1_RB"."TH. CUA DONG" )
      wire#w5
      Contact( "C#1_RB"."XA W_FD1" )
      Contact( "LUU TAY CEM1" )
      wire#w6
      I_Contact( "C#8_RD_REPORT".SAVE_REPORT )
      I_Contact( "PLC_BIT".RUN )
      Coil( "LUU_CAN TAY" )
   END_RUNG
   RUNG wire#w5
      Contact( "C#1_RB"."XA W_AP1" )
      Contact( "LUU TAY WAT1" )
   END_RUNG wire#w6
   RUNG wire#w5
      Contact( "C#1_RB"."XA W_SB1" )
      Contact( "LUU TAY WAT1" )
   END_RUNG wire#w6
   RUNG wire#powerrail
      Contact( "LUU_CAN TAY" )
   END_RUNG wire#w6
   RUNG wire#powerrail
      P_Contact(operand := "PLC_BIT".NTR_FU, bit := "P_MIXER_FU")
      Add(in1 := "C#7_RD_RUN".SMC_MIXER, in2 := 1.0, out => "C#7_RD_RUN".SMC_MIXER)
   END_RUNG
   // the same network as SCL:
   #_w1 := ((("C#7_RD_RUN".SMX_AP1 = "C#7_RD_RUN".SMX_FD1) OR ("C#4_WD_WEIGHT".SV_FD1 = 0.0)) AND ("C#7_RD_RUN".SMX_AP1 = "C#7_RD_RUN".SMX_AG1) AND ("C#7_RD_RUN".SMX_AP1 > "C#7_RD_RUN".SMC_MIXER) AND (("C#7_RD_RUN".SMX_AP1 = "C#7_RD_RUN".SMX_SB1) OR ("C#4_WD_WEIGHT".SV_SB1 = 0.0) OR ("C#4_WD_WEIGHT".SV_FD1 = 0.0))) OR ("LUU_CAN TAY" AND "C#1_RB"."MO CUA");
   IF #_w1 AND "C#2_WB"."SW_MAN/AUTO" THEN "PLC_BIT".NTR_FU := TRUE; END_IF;
   IF #_w1 THEN "C#8_RD_REPORT".SAVE_REPORT := TRUE; END_IF;
   IF "9.13_RESET_SAVE".OUT OR (NOT "C#2_WB"."SW_MAN/AUTO" AND "C#1_RB"."DONG CUA") OR "C#2_WB".F1_NN_RUN THEN
       "C#8_RD_REPORT".SAVE_REPORT := FALSE;
   END_IF;
   "LUU_CAN TAY" := ((NOT "C#2_WB"."SW_MAN/AUTO" AND "C#1_RB"."TH. CUA DONG" AND (("C#1_RB"."XA W_FD1" AND "LUU TAY CEM1") OR ("C#1_RB"."XA W_AP1" AND "LUU TAY WAT1") OR ("C#1_RB"."XA W_SB1" AND "LUU TAY WAT1"))) OR "LUU_CAN TAY") AND NOT "C#8_RD_REPORT".SAVE_REPORT AND NOT "PLC_BIT".RUN;
   #_w2 := "PLC_BIT".NTR_FU AND NOT "P_MIXER_FU";   // rising edge of "PLC_BIT".NTR_FU
   "P_MIXER_FU" := "PLC_BIT".NTR_FU;
   IF #_w2 THEN "C#7_RD_RUN".SMC_MIXER := "C#7_RD_RUN".SMC_MIXER + 1.0; END_IF;
END_REGION

REGION Network 14: QUA TRÌNH NẠP LIỆU NỒI TRỘN
   RUNG wire#powerrail
      "5. QUA TRINH NAP LIEU"(XA_PTG => "C#1_RB"."XA W_AG1", XA_CEM1 => "C#1_RB"."XA W_FD1", XA_CEM2 => "AlwaysFALSE", XA_WAT1 => "C#1_RB"."XA W_AP1", XA_WAT2 => "AlwaysFALSE", XA_ADD1 => "C#1_RB"."XA W_SB1", XA_ADD2 => "AlwaysFALSE")
   END_RUNG
   // the same network as SCL:
   "5. QUA TRINH NAP LIEU"(XA_PTG => "C#1_RB"."XA W_AG1",
                           XA_CEM1 => "C#1_RB"."XA W_FD1",
                           XA_CEM2 => "AlwaysFALSE",
                           XA_WAT1 => "C#1_RB"."XA W_AP1",
                           XA_WAT2 => "AlwaysFALSE",
                           XA_ADD1 => "C#1_RB"."XA W_SB1",
                           XA_ADD2 => "AlwaysFALSE");
END_REGION

REGION Network 15: RESET NAP LIEU VA THOI GIAN TRE NAP SAU PTG
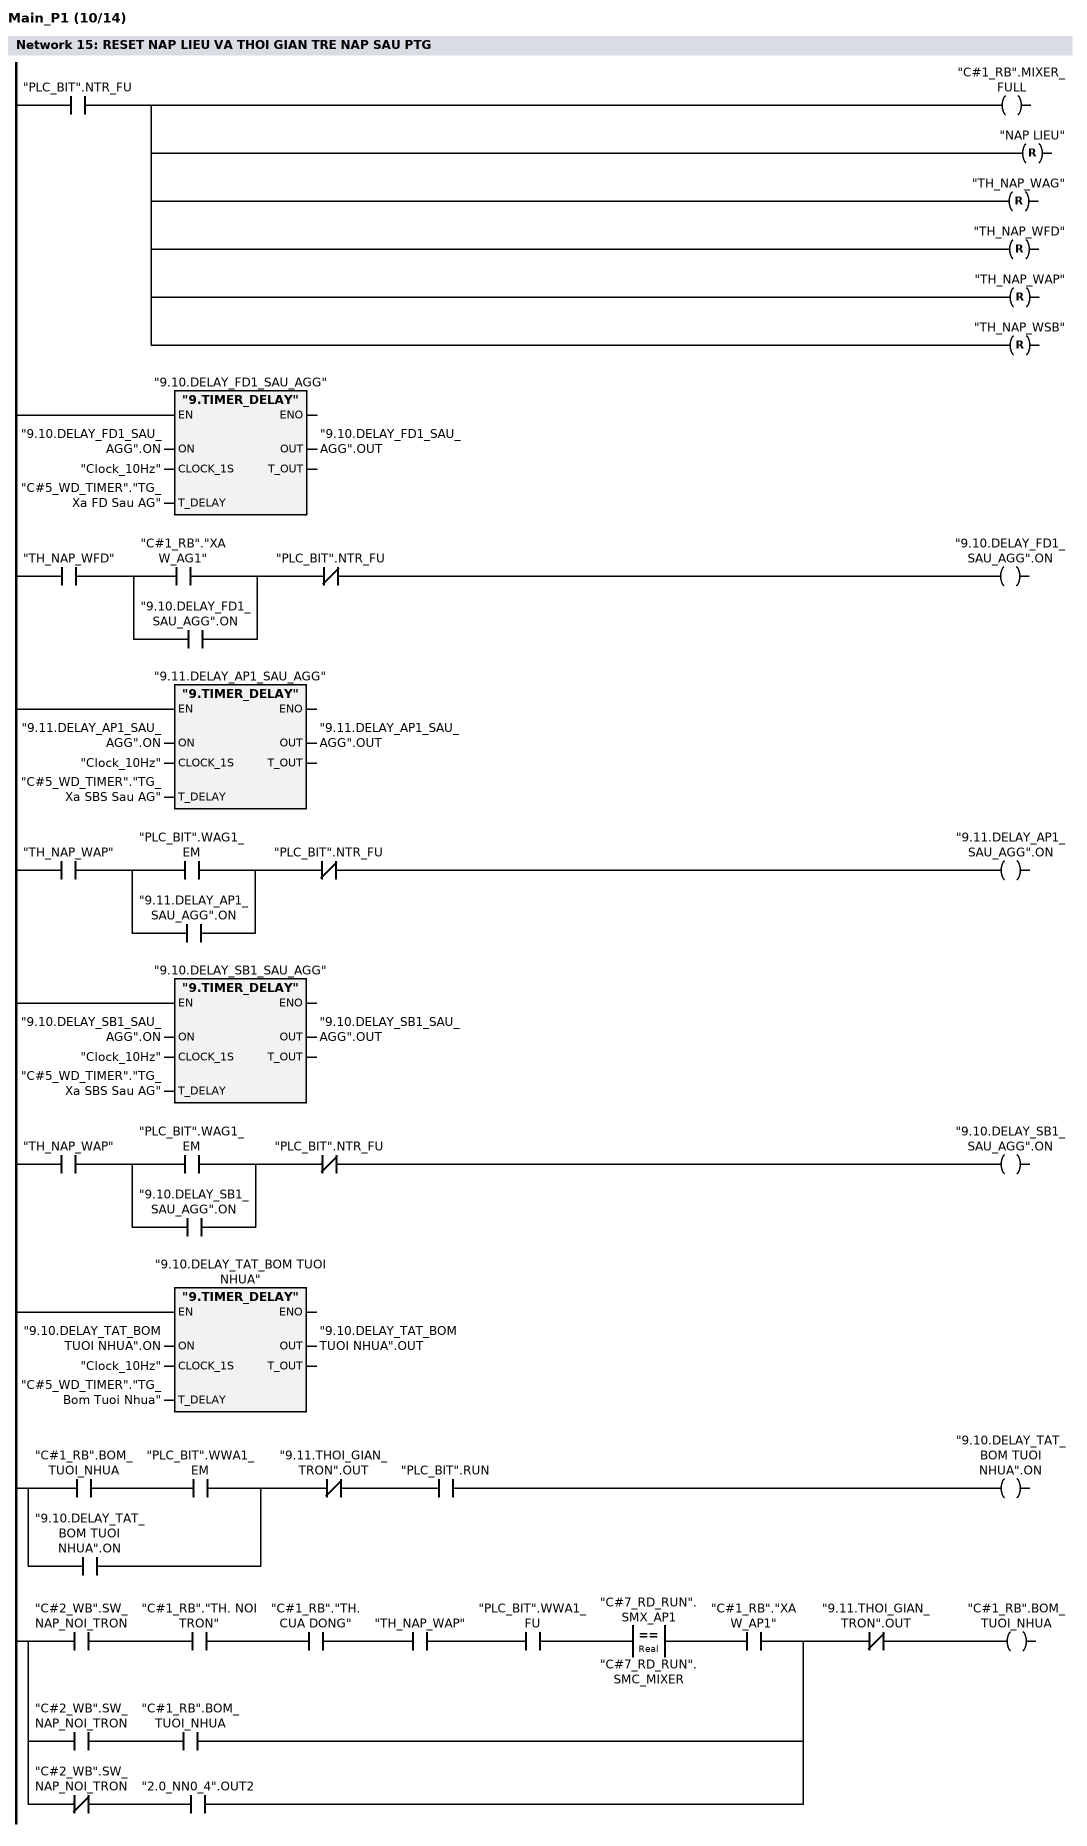
   RUNG wire#powerrail
      Contact( "PLC_BIT".NTR_FU )
      wire#w1
      Coil( "C#1_RB".MIXER_FULL )
   END_RUNG
   RUNG wire#w1
      R_Coil( "NAP LIEU" )
   END_RUNG
   RUNG wire#w1
      R_Coil( "TH_NAP_WAG" )
   END_RUNG
   RUNG wire#w1
      R_Coil( "TH_NAP_WFD" )
   END_RUNG
   RUNG wire#w1
      R_Coil( "TH_NAP_WAP" )
   END_RUNG
   RUNG wire#w1
      R_Coil( "TH_NAP_WSB" )
   END_RUNG
   RUNG wire#powerrail
      "9.10.DELAY_FD1_SAU_AGG"(ON := "9.10.DELAY_FD1_SAU_AGG".ON, CLOCK_1S := "Clock_10Hz", T_DELAY := "C#5_WD_TIMER"."TG_Xa FD Sau AG", OUT => "9.10.DELAY_FD1_SAU_AGG".OUT, T_OUT =>)
   END_RUNG
   RUNG wire#powerrail
      Contact( "TH_NAP_WFD" )
      wire#w2
      Contact( "C#1_RB"."XA W_AG1" )
      wire#w3
      I_Contact( "PLC_BIT".NTR_FU )
      Coil( "9.10.DELAY_FD1_SAU_AGG".ON )
   END_RUNG
   RUNG wire#w2
      Contact( "9.10.DELAY_FD1_SAU_AGG".ON )
   END_RUNG wire#w3
   RUNG wire#powerrail
      "9.11.DELAY_AP1_SAU_AGG"(ON := "9.11.DELAY_AP1_SAU_AGG".ON, CLOCK_1S := "Clock_10Hz", T_DELAY := "C#5_WD_TIMER"."TG_Xa SBS Sau AG", OUT => "9.11.DELAY_AP1_SAU_AGG".OUT, T_OUT =>)
   END_RUNG
   RUNG wire#powerrail
      Contact( "TH_NAP_WAP" )
      wire#w4
      Contact( "PLC_BIT".WAG1_EM )
      wire#w5
      I_Contact( "PLC_BIT".NTR_FU )
      Coil( "9.11.DELAY_AP1_SAU_AGG".ON )
   END_RUNG
   RUNG wire#w4
      Contact( "9.11.DELAY_AP1_SAU_AGG".ON )
   END_RUNG wire#w5
   RUNG wire#powerrail
      "9.10.DELAY_SB1_SAU_AGG"(ON := "9.10.DELAY_SB1_SAU_AGG".ON, CLOCK_1S := "Clock_10Hz", T_DELAY := "C#5_WD_TIMER"."TG_Xa SBS Sau AG", OUT => "9.10.DELAY_SB1_SAU_AGG".OUT, T_OUT =>)
   END_RUNG
   RUNG wire#powerrail
      Contact( "TH_NAP_WAP" )
      wire#w6
      Contact( "PLC_BIT".WAG1_EM )
      wire#w7
      I_Contact( "PLC_BIT".NTR_FU )
      Coil( "9.10.DELAY_SB1_SAU_AGG".ON )
   END_RUNG
   RUNG wire#w6
      Contact( "9.10.DELAY_SB1_SAU_AGG".ON )
   END_RUNG wire#w7
   RUNG wire#powerrail
      "9.10.DELAY_TAT_BOM TUOI NHUA"(ON := "9.10.DELAY_TAT_BOM TUOI NHUA".ON, CLOCK_1S := "Clock_10Hz", T_DELAY := "C#5_WD_TIMER"."TG_Bom Tuoi Nhua", OUT => "9.10.DELAY_TAT_BOM TUOI NHUA".OUT, T_OUT =>)
   END_RUNG
   RUNG wire#powerrail
      Contact( "C#1_RB".BOM_TUOI_NHUA )
      Contact( "PLC_BIT".WWA1_EM )
      wire#w8
      I_Contact( "9.11.THOI_GIAN_TRON".OUT )
      Contact( "PLC_BIT".RUN )
      Coil( "9.10.DELAY_TAT_BOM TUOI NHUA".ON )
   END_RUNG
   RUNG wire#powerrail
      Contact( "9.10.DELAY_TAT_BOM TUOI NHUA".ON )
   END_RUNG wire#w8
   RUNG wire#powerrail
      Contact( "C#2_WB".SW_NAP_NOI_TRON )
      Contact( "C#1_RB"."TH. NOI TRON" )
      Contact( "C#1_RB"."TH. CUA DONG" )
      Contact( "TH_NAP_WAP" )
      Contact( "PLC_BIT".WWA1_FU )
      { S7_Templates := "SrcType := Real" } EQ_Contact(in1 := "C#7_RD_RUN".SMX_AP1, in2 := "C#7_RD_RUN".SMC_MIXER)
      Contact( "C#1_RB"."XA W_AP1" )
      wire#w9
      I_Contact( "9.11.THOI_GIAN_TRON".OUT )
      Coil( "C#1_RB".BOM_TUOI_NHUA )
   END_RUNG
   RUNG wire#powerrail
      Contact( "C#2_WB".SW_NAP_NOI_TRON )
      Contact( "C#1_RB".BOM_TUOI_NHUA )
   END_RUNG wire#w9
   RUNG wire#powerrail
      I_Contact( "C#2_WB".SW_NAP_NOI_TRON )
      Contact( "2.0_NN0_4".OUT2 )
   END_RUNG wire#w9
   // the same network as SCL:
   "C#1_RB".MIXER_FULL := "PLC_BIT".NTR_FU;
   IF "PLC_BIT".NTR_FU THEN
       "NAP LIEU" := FALSE;
       "TH_NAP_WAG" := FALSE;
       "TH_NAP_WFD" := FALSE;
       "TH_NAP_WAP" := FALSE;
       "TH_NAP_WSB" := FALSE;
   END_IF;
   "9.10.DELAY_FD1_SAU_AGG"(ON := "9.10.DELAY_FD1_SAU_AGG".ON,   // "9.TIMER_DELAY"
                           CLOCK_1S := "Clock_10Hz",
                           T_DELAY := "C#5_WD_TIMER"."TG_Xa FD Sau AG",
                           OUT => "9.10.DELAY_FD1_SAU_AGG".OUT);
   "9.10.DELAY_FD1_SAU_AGG".ON := "TH_NAP_WFD" AND ("C#1_RB"."XA W_AG1" OR "9.10.DELAY_FD1_SAU_AGG".ON) AND NOT "PLC_BIT".NTR_FU;
   "9.11.DELAY_AP1_SAU_AGG"(ON := "9.11.DELAY_AP1_SAU_AGG".ON,   // "9.TIMER_DELAY"
                           CLOCK_1S := "Clock_10Hz",
                           T_DELAY := "C#5_WD_TIMER"."TG_Xa SBS Sau AG",
                           OUT => "9.11.DELAY_AP1_SAU_AGG".OUT);
   "9.11.DELAY_AP1_SAU_AGG".ON := "TH_NAP_WAP" AND ("PLC_BIT".WAG1_EM OR "9.11.DELAY_AP1_SAU_AGG".ON) AND NOT "PLC_BIT".NTR_FU;
   "9.10.DELAY_SB1_SAU_AGG"(ON := "9.10.DELAY_SB1_SAU_AGG".ON,   // "9.TIMER_DELAY"
                           CLOCK_1S := "Clock_10Hz",
                           T_DELAY := "C#5_WD_TIMER"."TG_Xa SBS Sau AG",
                           OUT => "9.10.DELAY_SB1_SAU_AGG".OUT);
   "9.10.DELAY_SB1_SAU_AGG".ON := "TH_NAP_WAP" AND ("PLC_BIT".WAG1_EM OR "9.10.DELAY_SB1_SAU_AGG".ON) AND NOT "PLC_BIT".NTR_FU;
   "9.10.DELAY_TAT_BOM TUOI NHUA"(ON := "9.10.DELAY_TAT_BOM TUOI NHUA".ON,   // "9.TIMER_DELAY"
                           CLOCK_1S := "Clock_10Hz",
                           T_DELAY := "C#5_WD_TIMER"."TG_Bom Tuoi Nhua",
                           OUT => "9.10.DELAY_TAT_BOM TUOI NHUA".OUT);
   "9.10.DELAY_TAT_BOM TUOI NHUA".ON := (("C#1_RB".BOM_TUOI_NHUA AND "PLC_BIT".WWA1_EM) OR "9.10.DELAY_TAT_BOM TUOI NHUA".ON) AND NOT "9.11.THOI_GIAN_TRON".OUT AND "PLC_BIT".RUN;
   "C#1_RB".BOM_TUOI_NHUA := (("C#2_WB".SW_NAP_NOI_TRON AND "C#1_RB"."TH. NOI TRON" AND "C#1_RB"."TH. CUA DONG" AND "TH_NAP_WAP" AND "PLC_BIT".WWA1_FU AND ("C#7_RD_RUN".SMX_AP1 = "C#7_RD_RUN".SMC_MIXER) AND "C#1_RB"."XA W_AP1") OR ("C#2_WB".SW_NAP_NOI_TRON AND "C#1_RB".BOM_TUOI_NHUA) OR (NOT "C#2_WB".SW_NAP_NOI_TRON AND "2.0_NN0_4".OUT2)) AND NOT "9.11.THOI_GIAN_TRON".OUT;
END_REGION

REGION Network 16: THOI GIAN TRON
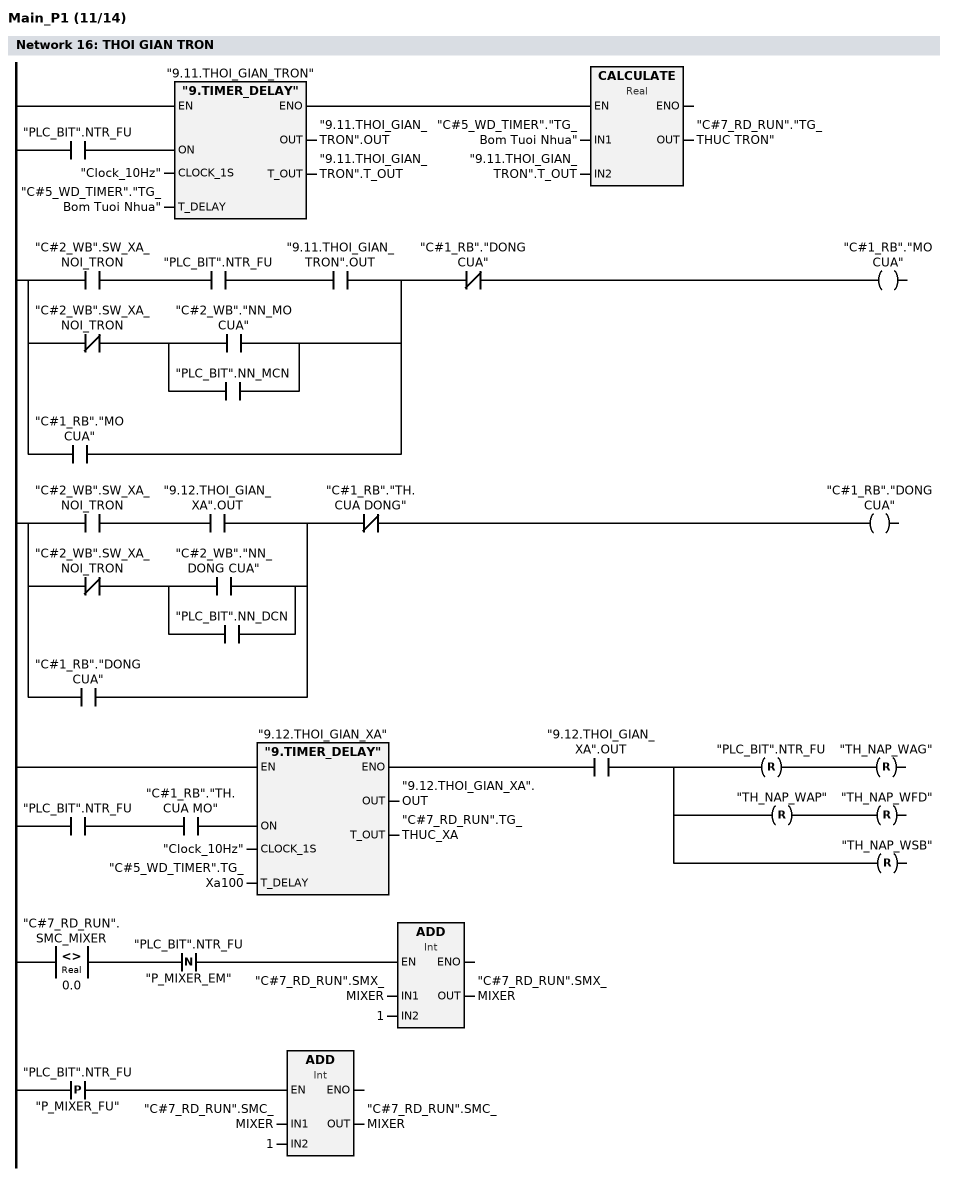
   RUNG wire#powerrail
      "9.11.THOI_GIAN_TRON"(ON := wire#w1, CLOCK_1S := "Clock_10Hz", T_DELAY := "C#5_WD_TIMER"."TG_Bom Tuoi Nhua", OUT => "9.11.THOI_GIAN_TRON".OUT, T_OUT => "9.11.THOI_GIAN_TRON".T_OUT)
      { S7_Templates := "SrcType := Real"; S7_Expression := "IN1-IN2" } Calculate(in1 := "C#5_WD_TIMER"."TG_Bom Tuoi Nhua", in2 := "9.11.THOI_GIAN_TRON".T_OUT, out => "C#7_RD_RUN"."TG_THUC TRON")
   END_RUNG
   RUNG wire#powerrail
      Contact( "PLC_BIT".NTR_FU )
   END_RUNG wire#w1
   RUNG wire#powerrail
      Contact( "C#2_WB".SW_XA_NOI_TRON )
      Contact( "PLC_BIT".NTR_FU )
      Contact( "9.11.THOI_GIAN_TRON".OUT )
      wire#w2
      I_Contact( "C#1_RB"."DONG CUA" )
      Coil( "C#1_RB"."MO CUA" )
   END_RUNG
   RUNG wire#powerrail
      I_Contact( "C#2_WB".SW_XA_NOI_TRON )
      wire#w3
      Contact( "C#2_WB"."NN_MO CUA" )
   END_RUNG wire#w2
   RUNG wire#w3
      Contact( "PLC_BIT".NN_MCN )
   END_RUNG wire#w2
   RUNG wire#powerrail
      Contact( "C#1_RB"."MO CUA" )
   END_RUNG wire#w2
   RUNG wire#powerrail
      Contact( "C#2_WB".SW_XA_NOI_TRON )
      Contact( "9.12.THOI_GIAN_XA".OUT )
      wire#w4
      I_Contact( "C#1_RB"."TH. CUA DONG" )
      Coil( "C#1_RB"."DONG CUA" )
   END_RUNG
   RUNG wire#powerrail
      I_Contact( "C#2_WB".SW_XA_NOI_TRON )
      wire#w5
      Contact( "C#2_WB"."NN_DONG CUA" )
   END_RUNG wire#w4
   RUNG wire#w5
      Contact( "PLC_BIT".NN_DCN )
   END_RUNG wire#w4
   RUNG wire#powerrail
      Contact( "C#1_RB"."DONG CUA" )
   END_RUNG wire#w4
   RUNG wire#powerrail
      "9.12.THOI_GIAN_XA"(ON := wire#w6, CLOCK_1S := "Clock_10Hz", T_DELAY := "C#5_WD_TIMER".TG_Xa100, OUT => "9.12.THOI_GIAN_XA".OUT, T_OUT => "C#7_RD_RUN".TG_THUC_XA)
      Contact( "9.12.THOI_GIAN_XA".OUT )
      wire#w7
      R_Coil( "PLC_BIT".NTR_FU )
      R_Coil( "TH_NAP_WAG" )
   END_RUNG
   RUNG wire#powerrail
      Contact( "PLC_BIT".NTR_FU )
      Contact( "C#1_RB"."TH. CUA MO" )
   END_RUNG wire#w6
   RUNG wire#w7
      R_Coil( "TH_NAP_WAP" )
      R_Coil( "TH_NAP_WFD" )
   END_RUNG
   RUNG wire#w7
      R_Coil( "TH_NAP_WSB" )
   END_RUNG
   RUNG wire#powerrail
      { S7_Templates := "SrcType := Real" } NE_Contact(in1 := "C#7_RD_RUN".SMC_MIXER, in2 := 0.0)
      N_Contact(operand := "PLC_BIT".NTR_FU, bit := "P_MIXER_EM")
      { S7_Templates := "SrcType := Int" } Add(in1 := "C#7_RD_RUN".SMX_MIXER, in2 := 1, out => "C#7_RD_RUN".SMX_MIXER)
   END_RUNG
   RUNG wire#powerrail
      P_Contact(operand := "PLC_BIT".NTR_FU, bit := "P_MIXER_FU")
      { S7_Templates := "SrcType := Int" } Add(in1 := "C#7_RD_RUN".SMC_MIXER, in2 := 1, out => "C#7_RD_RUN".SMC_MIXER)
   END_RUNG
   // the same network as SCL:
   "9.11.THOI_GIAN_TRON"(ON := "PLC_BIT".NTR_FU,   // "9.TIMER_DELAY"
                         CLOCK_1S := "Clock_10Hz",
                         T_DELAY := "C#5_WD_TIMER"."TG_Bom Tuoi Nhua",
                         OUT => "9.11.THOI_GIAN_TRON".OUT,
                         T_OUT => "9.11.THOI_GIAN_TRON".T_OUT,
                         ENO => #_w1);
   IF #_w1 THEN
       "C#7_RD_RUN"."TG_THUC TRON" := "C#5_WD_TIMER"."TG_Bom Tuoi Nhua"-"9.11.THOI_GIAN_TRON".T_OUT;
   END_IF;
   "C#1_RB"."MO CUA" := (("C#2_WB".SW_XA_NOI_TRON AND "PLC_BIT".NTR_FU AND "9.11.THOI_GIAN_TRON".OUT) OR (NOT "C#2_WB".SW_XA_NOI_TRON AND ("C#2_WB"."NN_MO CUA" OR "PLC_BIT".NN_MCN)) OR "C#1_RB"."MO CUA") AND NOT "C#1_RB"."DONG CUA";
   "C#1_RB"."DONG CUA" := (("C#2_WB".SW_XA_NOI_TRON AND "9.12.THOI_GIAN_XA".OUT) OR (NOT "C#2_WB".SW_XA_NOI_TRON AND ("C#2_WB"."NN_DONG CUA" OR "PLC_BIT".NN_DCN)) OR "C#1_RB"."DONG CUA") AND NOT "C#1_RB"."TH. CUA DONG";
   "9.12.THOI_GIAN_XA"(ON := "PLC_BIT".NTR_FU AND "C#1_RB"."TH. CUA MO",   // "9.TIMER_DELAY"
                       CLOCK_1S := "Clock_10Hz",
                       T_DELAY := "C#5_WD_TIMER".TG_Xa100,
                       OUT => "9.12.THOI_GIAN_XA".OUT,
                       T_OUT => "C#7_RD_RUN".TG_THUC_XA,
                       ENO => #_w2);
   IF #_w2 AND "9.12.THOI_GIAN_XA".OUT THEN
       "PLC_BIT".NTR_FU := FALSE;
       "TH_NAP_WAG" := FALSE;
       "TH_NAP_WAP" := FALSE;
       "TH_NAP_WFD" := FALSE;
       "TH_NAP_WSB" := FALSE;
   END_IF;
   #_w3 := ("C#7_RD_RUN".SMC_MIXER <> 0.0) AND NOT "PLC_BIT".NTR_FU AND "P_MIXER_EM";   // falling edge of "PLC_BIT".NTR_FU
   "P_MIXER_EM" := "PLC_BIT".NTR_FU;
   IF #_w3 THEN "C#7_RD_RUN".SMX_MIXER := "C#7_RD_RUN".SMX_MIXER + 1; END_IF;
   #_w4 := "PLC_BIT".NTR_FU AND NOT "P_MIXER_FU";   // rising edge of "PLC_BIT".NTR_FU
   "P_MIXER_FU" := "PLC_BIT".NTR_FU;
   IF #_w4 THEN "C#7_RD_RUN".SMC_MIXER := "C#7_RD_RUN".SMC_MIXER + 1; END_IF;
END_REGION

REGION Network 17: TEST SAVE DATA
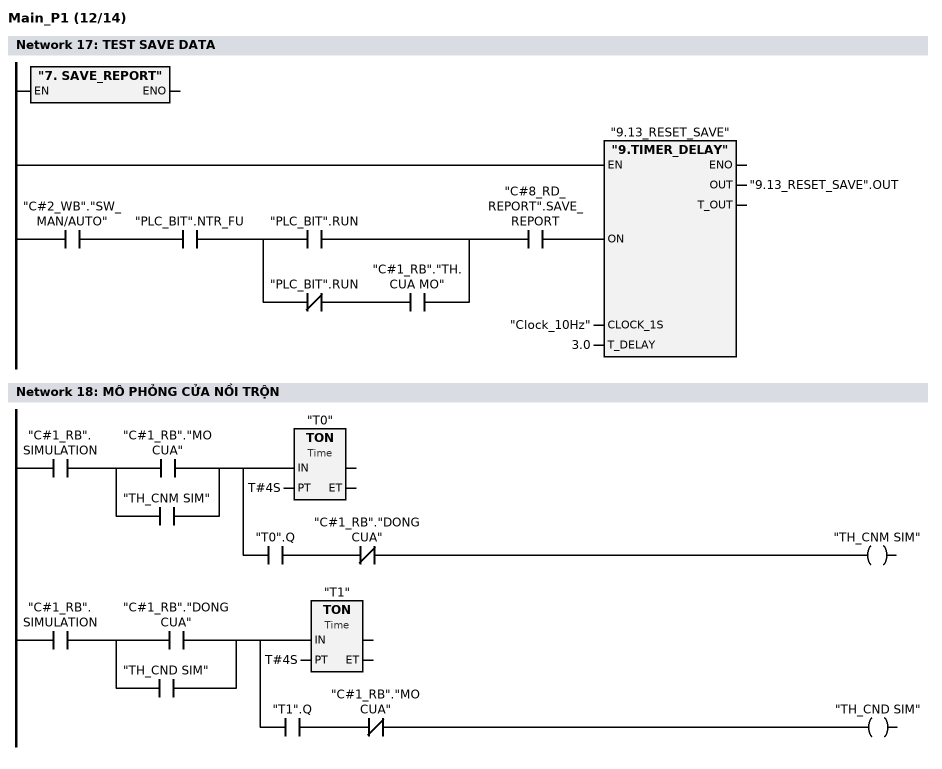
   RUNG wire#powerrail
      "7. SAVE_REPORT"()
   END_RUNG
   RUNG wire#powerrail
      "9.13_RESET_SAVE"(ON := wire#w3, CLOCK_1S := "Clock_10Hz", T_DELAY := 3.0, OUT => "9.13_RESET_SAVE".OUT, T_OUT =>)
   END_RUNG
   RUNG wire#powerrail
      Contact( "C#2_WB"."SW_MAN/AUTO" )
      Contact( "PLC_BIT".NTR_FU )
      wire#w1
      Contact( "PLC_BIT".RUN )
      wire#w2
      Contact( "C#8_RD_REPORT".SAVE_REPORT )
   END_RUNG wire#w3
   RUNG wire#w1
      I_Contact( "PLC_BIT".RUN )
      Contact( "C#1_RB"."TH. CUA MO" )
   END_RUNG wire#w2
   // the same network as SCL:
   "7. SAVE_REPORT"();
   "9.13_RESET_SAVE"(ON := "C#2_WB"."SW_MAN/AUTO" AND "PLC_BIT".NTR_FU AND ("PLC_BIT".RUN OR (NOT "PLC_BIT".RUN AND "C#1_RB"."TH. CUA MO")) AND "C#8_RD_REPORT".SAVE_REPORT,   // "9.TIMER_DELAY"
                     CLOCK_1S := "Clock_10Hz",
                     T_DELAY := 3.0,
                     OUT => "9.13_RESET_SAVE".OUT);
END_REGION

REGION Network 18: MÔ PHỎNG CỬA NỒI TRỘN
   RUNG wire#powerrail
      Contact( "C#1_RB".SIMULATION )
      wire#w1
      Contact( "C#1_RB"."MO CUA" )
      wire#w2
      { S7_Templates := "time_type := Time" } "T0".TON(pt := T#4S, et =>)
   END_RUNG
   RUNG wire#w1
      Contact( "TH_CNM SIM" )
   END_RUNG wire#w2
   RUNG wire#w2
      Contact( "T0".Q )
      I_Contact( "C#1_RB"."DONG CUA" )
      Coil( "TH_CNM SIM" )
   END_RUNG
   RUNG wire#powerrail
      Contact( "C#1_RB".SIMULATION )
      wire#w3
      Contact( "C#1_RB"."DONG CUA" )
      wire#w4
      { S7_Templates := "time_type := Time" } "T1".TON(pt := T#4S, et =>)
   END_RUNG
   RUNG wire#w3
      Contact( "TH_CND SIM" )
   END_RUNG wire#w4
   RUNG wire#w4
      Contact( "T1".Q )
      I_Contact( "C#1_RB"."MO CUA" )
      Coil( "TH_CND SIM" )
   END_RUNG
   // the same network as SCL:
   #_w1 := "C#1_RB".SIMULATION AND ("C#1_RB"."MO CUA" OR "TH_CNM SIM");
   "T0".TON(IN := #_w1, PT := T#4S);
   "TH_CNM SIM" := #_w1 AND "T0".Q AND NOT "C#1_RB"."DONG CUA";
   #_w2 := "C#1_RB".SIMULATION AND ("C#1_RB"."DONG CUA" OR "TH_CND SIM");
   "T1".TON(IN := #_w2, PT := T#4S);
   "TH_CND SIM" := #_w2 AND "T1".Q AND NOT "C#1_RB"."MO CUA";
END_REGION

REGION Network 19: CHẾ ĐỘ XẢ LIỆU
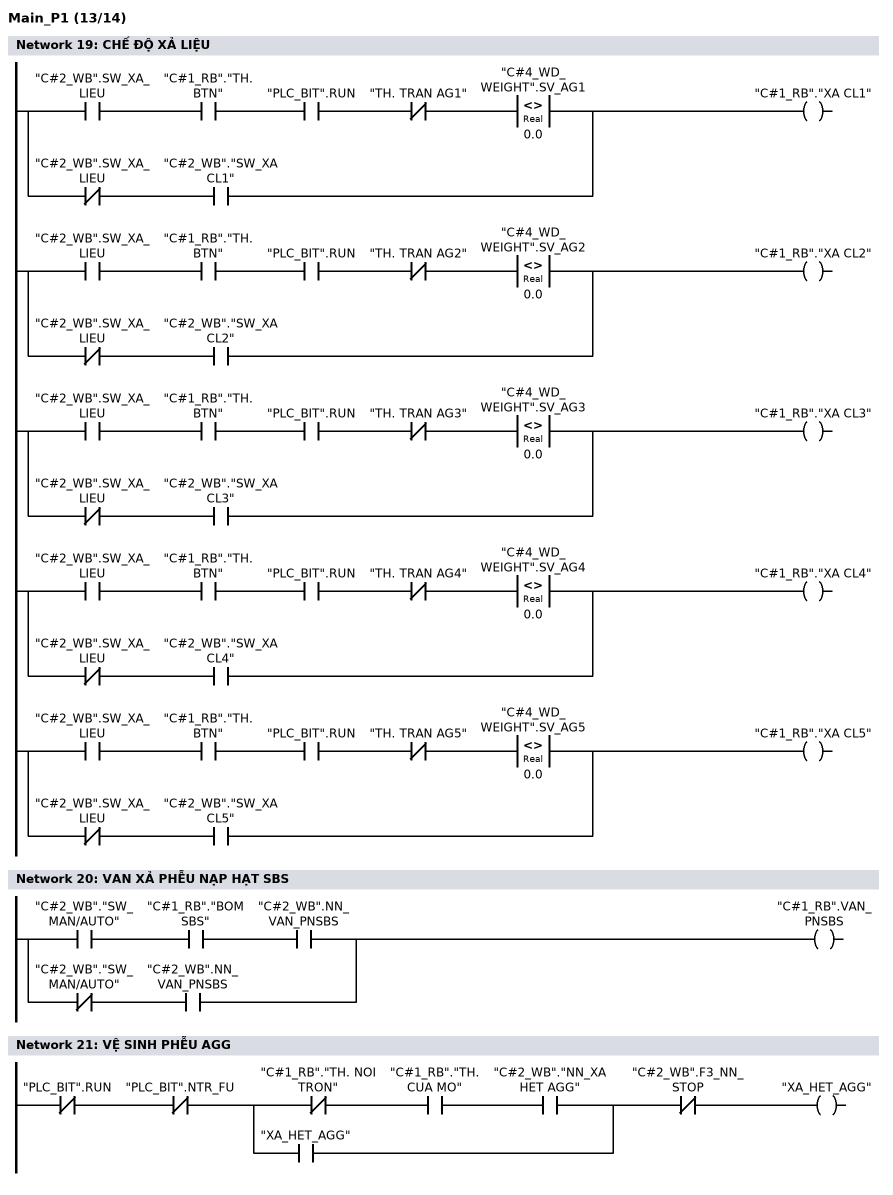
   RUNG wire#powerrail
      Contact( "C#2_WB".SW_XA_LIEU )
      Contact( "C#1_RB"."TH. BTN" )
      Contact( "PLC_BIT".RUN )
      I_Contact( "TH. TRAN AG1" )
      { S7_Templates := "SrcType := Real" } NE_Contact(in1 := "C#4_WD_WEIGHT".SV_AG1, in2 := 0.0)
      wire#w1
      Coil( "C#1_RB"."XA CL1" )
   END_RUNG
   RUNG wire#powerrail
      I_Contact( "C#2_WB".SW_XA_LIEU )
      Contact( "C#2_WB"."SW_XA CL1" )
   END_RUNG wire#w1
   RUNG wire#powerrail
      Contact( "C#2_WB".SW_XA_LIEU )
      Contact( "C#1_RB"."TH. BTN" )
      Contact( "PLC_BIT".RUN )
      I_Contact( "TH. TRAN AG2" )
      { S7_Templates := "SrcType := Real" } NE_Contact(in1 := "C#4_WD_WEIGHT".SV_AG2, in2 := 0.0)
      wire#w2
      Coil( "C#1_RB"."XA CL2" )
   END_RUNG
   RUNG wire#powerrail
      I_Contact( "C#2_WB".SW_XA_LIEU )
      Contact( "C#2_WB"."SW_XA CL2" )
   END_RUNG wire#w2
   RUNG wire#powerrail
      Contact( "C#2_WB".SW_XA_LIEU )
      Contact( "C#1_RB"."TH. BTN" )
      Contact( "PLC_BIT".RUN )
      I_Contact( "TH. TRAN AG3" )
      { S7_Templates := "SrcType := Real" } NE_Contact(in1 := "C#4_WD_WEIGHT".SV_AG3, in2 := 0.0)
      wire#w3
      Coil( "C#1_RB"."XA CL3" )
   END_RUNG
   RUNG wire#powerrail
      I_Contact( "C#2_WB".SW_XA_LIEU )
      Contact( "C#2_WB"."SW_XA CL3" )
   END_RUNG wire#w3
   RUNG wire#powerrail
      Contact( "C#2_WB".SW_XA_LIEU )
      Contact( "C#1_RB"."TH. BTN" )
      Contact( "PLC_BIT".RUN )
      I_Contact( "TH. TRAN AG4" )
      { S7_Templates := "SrcType := Real" } NE_Contact(in1 := "C#4_WD_WEIGHT".SV_AG4, in2 := 0.0)
      wire#w4
      Coil( "C#1_RB"."XA CL4" )
   END_RUNG
   RUNG wire#powerrail
      I_Contact( "C#2_WB".SW_XA_LIEU )
      Contact( "C#2_WB"."SW_XA CL4" )
   END_RUNG wire#w4
   RUNG wire#powerrail
      Contact( "C#2_WB".SW_XA_LIEU )
      Contact( "C#1_RB"."TH. BTN" )
      Contact( "PLC_BIT".RUN )
      I_Contact( "TH. TRAN AG5" )
      { S7_Templates := "SrcType := Real" } NE_Contact(in1 := "C#4_WD_WEIGHT".SV_AG5, in2 := 0.0)
      wire#w5
      Coil( "C#1_RB"."XA CL5" )
   END_RUNG
   RUNG wire#powerrail
      I_Contact( "C#2_WB".SW_XA_LIEU )
      Contact( "C#2_WB"."SW_XA CL5" )
   END_RUNG wire#w5
   // the same network as SCL:
   "C#1_RB"."XA CL1" := ("C#2_WB".SW_XA_LIEU AND "C#1_RB"."TH. BTN" AND "PLC_BIT".RUN AND NOT "TH. TRAN AG1" AND ("C#4_WD_WEIGHT".SV_AG1 <> 0.0)) OR (NOT "C#2_WB".SW_XA_LIEU AND "C#2_WB"."SW_XA CL1");
   "C#1_RB"."XA CL2" := ("C#2_WB".SW_XA_LIEU AND "C#1_RB"."TH. BTN" AND "PLC_BIT".RUN AND NOT "TH. TRAN AG2" AND ("C#4_WD_WEIGHT".SV_AG2 <> 0.0)) OR (NOT "C#2_WB".SW_XA_LIEU AND "C#2_WB"."SW_XA CL2");
   "C#1_RB"."XA CL3" := ("C#2_WB".SW_XA_LIEU AND "C#1_RB"."TH. BTN" AND "PLC_BIT".RUN AND NOT "TH. TRAN AG3" AND ("C#4_WD_WEIGHT".SV_AG3 <> 0.0)) OR (NOT "C#2_WB".SW_XA_LIEU AND "C#2_WB"."SW_XA CL3");
   "C#1_RB"."XA CL4" := ("C#2_WB".SW_XA_LIEU AND "C#1_RB"."TH. BTN" AND "PLC_BIT".RUN AND NOT "TH. TRAN AG4" AND ("C#4_WD_WEIGHT".SV_AG4 <> 0.0)) OR (NOT "C#2_WB".SW_XA_LIEU AND "C#2_WB"."SW_XA CL4");
   "C#1_RB"."XA CL5" := ("C#2_WB".SW_XA_LIEU AND "C#1_RB"."TH. BTN" AND "PLC_BIT".RUN AND NOT "TH. TRAN AG5" AND ("C#4_WD_WEIGHT".SV_AG5 <> 0.0)) OR (NOT "C#2_WB".SW_XA_LIEU AND "C#2_WB"."SW_XA CL5");
END_REGION

REGION Network 20: VAN XẢ PHỄU NẠP HẠT SBS
   RUNG wire#powerrail
      Contact( "C#2_WB"."SW_MAN/AUTO" )
      Contact( "C#1_RB"."BOM SBS" )
      Contact( "C#2_WB".NN_VAN_PNSBS )
      wire#w1
      Coil( "C#1_RB".VAN_PNSBS )
   END_RUNG
   RUNG wire#powerrail
      I_Contact( "C#2_WB"."SW_MAN/AUTO" )
      Contact( "C#2_WB".NN_VAN_PNSBS )
   END_RUNG wire#w1
   // the same network as SCL:
   "C#1_RB".VAN_PNSBS := ("C#2_WB"."SW_MAN/AUTO" AND "C#1_RB"."BOM SBS" AND "C#2_WB".NN_VAN_PNSBS) OR (NOT "C#2_WB"."SW_MAN/AUTO" AND "C#2_WB".NN_VAN_PNSBS);
END_REGION

REGION Network 21: VỆ SINH PHỄU AGG
   RUNG wire#powerrail
      I_Contact( "PLC_BIT".RUN )
      I_Contact( "PLC_BIT".NTR_FU )
      wire#w1
      I_Contact( "C#1_RB"."TH. NOI TRON" )
      Contact( "C#1_RB"."TH. CUA MO" )
      Contact( "C#2_WB"."NN_XA HET AGG" )
      wire#w2
      I_Contact( "C#2_WB".F3_NN_STOP )
      Coil( "XA_HET_AGG" )
   END_RUNG
   RUNG wire#w1
      Contact( "XA_HET_AGG" )
   END_RUNG wire#w2
   // the same network as SCL:
   "XA_HET_AGG" := NOT "PLC_BIT".RUN AND NOT "PLC_BIT".NTR_FU AND ((NOT "C#1_RB"."TH. NOI TRON" AND "C#1_RB"."TH. CUA MO" AND "C#2_WB"."NN_XA HET AGG") OR "XA_HET_AGG") AND NOT "C#2_WB".F3_NN_STOP;
END_REGION

REGION Network 22: RUNG PHEU COT LIEU
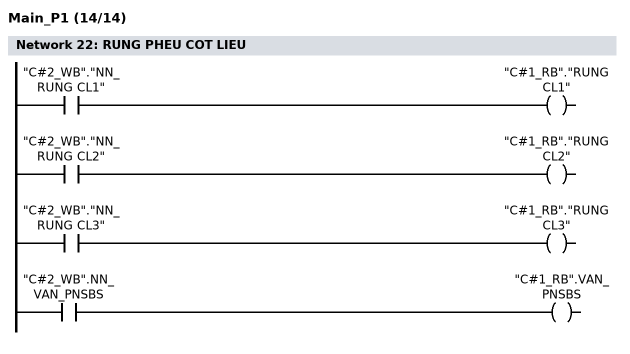
   RUNG wire#powerrail
      Contact( "C#2_WB"."NN_RUNG CL1" )
      Coil( "C#1_RB"."RUNG CL1" )
   END_RUNG
   RUNG wire#powerrail
      Contact( "C#2_WB"."NN_RUNG CL2" )
      Coil( "C#1_RB"."RUNG CL2" )
   END_RUNG
   RUNG wire#powerrail
      Contact( "C#2_WB"."NN_RUNG CL3" )
      Coil( "C#1_RB"."RUNG CL3" )
   END_RUNG
   RUNG wire#powerrail
      Contact( "C#2_WB".NN_VAN_PNSBS )
      Coil( "C#1_RB".VAN_PNSBS )
   END_RUNG
   // the same network as SCL:
   "C#1_RB"."RUNG CL1" := "C#2_WB"."NN_RUNG CL1";
   "C#1_RB"."RUNG CL2" := "C#2_WB"."NN_RUNG CL2";
   "C#1_RB"."RUNG CL3" := "C#2_WB"."NN_RUNG CL3";
   "C#1_RB".VAN_PNSBS := "C#2_WB".NN_VAN_PNSBS;
END_REGION
END_ORGANIZATION_BLOCK
